   // UNICODE_TO_GBK[39826] := 16#98FC;
   // UNICODE_TO_GBK[39827] := 16#EF95;
   // UNICODE_TO_GBK[39828] := 16#98FD;
   // UNICODE_TO_GBK[39829] := 16#EF96;
   // UNICODE_TO_GBK[39830] := 16#98FE;
   // UNICODE_TO_GBK[39831] := 16#EF97;
   // UNICODE_TO_GBK[39832] := 16#98FF;
   // UNICODE_TO_GBK[39833] := 16#EF98;
   // UNICODE_TO_GBK[39834] := 16#9900;
   // UNICODE_TO_GBK[39835] := 16#EF99;
   // UNICODE_TO_GBK[39836] := 16#9901;
   // UNICODE_TO_GBK[39837] := 16#EF9A;
   // UNICODE_TO_GBK[39838] := 16#9902;
   // UNICODE_TO_GBK[39839] := 16#EF9B;
   // UNICODE_TO_GBK[39840] := 16#9903;
   // UNICODE_TO_GBK[39841] := 16#EF9C;
   // UNICODE_TO_GBK[39842] := 16#9904;
   // UNICODE_TO_GBK[39843] := 16#EF9D;
   // UNICODE_TO_GBK[39844] := 16#9905;
   // UNICODE_TO_GBK[39845] := 16#EF9E;
   // UNICODE_TO_GBK[39846] := 16#9906;
   // UNICODE_TO_GBK[39847] := 16#EF9F;
   // UNICODE_TO_GBK[39848] := 16#9907;
   // UNICODE_TO_GBK[39849] := 16#EFA0;
   // UNICODE_TO_GBK[39850] := 16#9908;
   // UNICODE_TO_GBK[39851] := 16#F040;
   // UNICODE_TO_GBK[39852] := 16#9909;
   // UNICODE_TO_GBK[39853] := 16#F041;
   // UNICODE_TO_GBK[39854] := 16#990A;
   // UNICODE_TO_GBK[39855] := 16#F042;
   // UNICODE_TO_GBK[39856] := 16#990B;
   // UNICODE_TO_GBK[39857] := 16#F043;
   // UNICODE_TO_GBK[39858] := 16#990C;
   // UNICODE_TO_GBK[39859] := 16#F044;
   // UNICODE_TO_GBK[39860] := 16#990D;
   // UNICODE_TO_GBK[39861] := 16#F7D0;
   // UNICODE_TO_GBK[39862] := 16#990E;
   // UNICODE_TO_GBK[39863] := 16#F045;
   // UNICODE_TO_GBK[39864] := 16#990F;
   // UNICODE_TO_GBK[39865] := 16#F046;
   // UNICODE_TO_GBK[39866] := 16#9910;
   // UNICODE_TO_GBK[39867] := 16#B2CD;
   // UNICODE_TO_GBK[39868] := 16#9911;
   // UNICODE_TO_GBK[39869] := 16#F047;
   // UNICODE_TO_GBK[39870] := 16#9912;
   // UNICODE_TO_GBK[39871] := 16#F048;
   // UNICODE_TO_GBK[39872] := 16#9913;
   // UNICODE_TO_GBK[39873] := 16#F049;
   // UNICODE_TO_GBK[39874] := 16#9914;
   // UNICODE_TO_GBK[39875] := 16#F04A;
   // UNICODE_TO_GBK[39876] := 16#9915;
   // UNICODE_TO_GBK[39877] := 16#F04B;
   // UNICODE_TO_GBK[39878] := 16#9916;
   // UNICODE_TO_GBK[39879] := 16#F04C;
   // UNICODE_TO_GBK[39880] := 16#9917;
   // UNICODE_TO_GBK[39881] := 16#F04D;
   // UNICODE_TO_GBK[39882] := 16#9918;
   // UNICODE_TO_GBK[39883] := 16#F04E;
   // UNICODE_TO_GBK[39884] := 16#9919;
   // UNICODE_TO_GBK[39885] := 16#F04F;
   // UNICODE_TO_GBK[39886] := 16#991A;
   // UNICODE_TO_GBK[39887] := 16#F050;
   // UNICODE_TO_GBK[39888] := 16#991B;
   // UNICODE_TO_GBK[39889] := 16#F051;
   // UNICODE_TO_GBK[39890] := 16#991C;
   // UNICODE_TO_GBK[39891] := 16#F052;
   // UNICODE_TO_GBK[39892] := 16#991D;
   // UNICODE_TO_GBK[39893] := 16#F053;
   // UNICODE_TO_GBK[39894] := 16#991E;
   // UNICODE_TO_GBK[39895] := 16#F054;
   // UNICODE_TO_GBK[39896] := 16#991F;
   // UNICODE_TO_GBK[39897] := 16#F055;
   // UNICODE_TO_GBK[39898] := 16#9920;
   // UNICODE_TO_GBK[39899] := 16#F056;
   // UNICODE_TO_GBK[39900] := 16#9921;
   // UNICODE_TO_GBK[39901] := 16#F057;
   // UNICODE_TO_GBK[39902] := 16#9922;
   // UNICODE_TO_GBK[39903] := 16#F058;
   // UNICODE_TO_GBK[39904] := 16#9923;
   // UNICODE_TO_GBK[39905] := 16#F059;
   // UNICODE_TO_GBK[39906] := 16#9924;
   // UNICODE_TO_GBK[39907] := 16#F05A;
   // UNICODE_TO_GBK[39908] := 16#9925;
   // UNICODE_TO_GBK[39909] := 16#F05B;
   // UNICODE_TO_GBK[39910] := 16#9926;
   // UNICODE_TO_GBK[39911] := 16#F05C;
   // UNICODE_TO_GBK[39912] := 16#9927;
   // UNICODE_TO_GBK[39913] := 16#F05D;
   // UNICODE_TO_GBK[39914] := 16#9928;
   // UNICODE_TO_GBK[39915] := 16#F05E;
   // UNICODE_TO_GBK[39916] := 16#9929;
   // UNICODE_TO_GBK[39917] := 16#F05F;
   // UNICODE_TO_GBK[39918] := 16#992A;
   // UNICODE_TO_GBK[39919] := 16#F060;
   // UNICODE_TO_GBK[39920] := 16#992B;
   // UNICODE_TO_GBK[39921] := 16#F061;
   // UNICODE_TO_GBK[39922] := 16#992C;
   // UNICODE_TO_GBK[39923] := 16#F062;
   // UNICODE_TO_GBK[39924] := 16#992D;
   // UNICODE_TO_GBK[39925] := 16#F063;
   // UNICODE_TO_GBK[39926] := 16#992E;
   // UNICODE_TO_GBK[39927] := 16#F7D1;
   // UNICODE_TO_GBK[39928] := 16#992F;
   // UNICODE_TO_GBK[39929] := 16#F064;
   // UNICODE_TO_GBK[39930] := 16#9930;
   // UNICODE_TO_GBK[39931] := 16#F065;
   // UNICODE_TO_GBK[39932] := 16#9931;
   // UNICODE_TO_GBK[39933] := 16#F066;
   // UNICODE_TO_GBK[39934] := 16#9932;
   // UNICODE_TO_GBK[39935] := 16#F067;
   // UNICODE_TO_GBK[39936] := 16#9933;
   // UNICODE_TO_GBK[39937] := 16#F068;
   // UNICODE_TO_GBK[39938] := 16#9934;
   // UNICODE_TO_GBK[39939] := 16#F069;
   // UNICODE_TO_GBK[39940] := 16#9935;
   // UNICODE_TO_GBK[39941] := 16#F06A;
   // UNICODE_TO_GBK[39942] := 16#9936;
   // UNICODE_TO_GBK[39943] := 16#F06B;
   // UNICODE_TO_GBK[39944] := 16#9937;
   // UNICODE_TO_GBK[39945] := 16#F06C;
   // UNICODE_TO_GBK[39946] := 16#9938;
   // UNICODE_TO_GBK[39947] := 16#F06D;
   // UNICODE_TO_GBK[39948] := 16#9939;
   // UNICODE_TO_GBK[39949] := 16#F06E;
   // UNICODE_TO_GBK[39950] := 16#993A;
   // UNICODE_TO_GBK[39951] := 16#F06F;
   // UNICODE_TO_GBK[39952] := 16#993B;
   // UNICODE_TO_GBK[39953] := 16#F070;
   // UNICODE_TO_GBK[39954] := 16#993C;
   // UNICODE_TO_GBK[39955] := 16#F071;
   // UNICODE_TO_GBK[39956] := 16#993D;
   // UNICODE_TO_GBK[39957] := 16#F072;
   // UNICODE_TO_GBK[39958] := 16#993E;
   // UNICODE_TO_GBK[39959] := 16#F073;
   // UNICODE_TO_GBK[39960] := 16#993F;
   // UNICODE_TO_GBK[39961] := 16#F074;
   // UNICODE_TO_GBK[39962] := 16#9940;
   // UNICODE_TO_GBK[39963] := 16#F075;
   // UNICODE_TO_GBK[39964] := 16#9941;
   // UNICODE_TO_GBK[39965] := 16#F076;
   // UNICODE_TO_GBK[39966] := 16#9942;
   // UNICODE_TO_GBK[39967] := 16#F077;
   // UNICODE_TO_GBK[39968] := 16#9943;
   // UNICODE_TO_GBK[39969] := 16#F078;
   // UNICODE_TO_GBK[39970] := 16#9944;
   // UNICODE_TO_GBK[39971] := 16#F079;
   // UNICODE_TO_GBK[39972] := 16#9945;
   // UNICODE_TO_GBK[39973] := 16#F07A;
   // UNICODE_TO_GBK[39974] := 16#9946;
   // UNICODE_TO_GBK[39975] := 16#F07B;
   // UNICODE_TO_GBK[39976] := 16#9947;
   // UNICODE_TO_GBK[39977] := 16#F07C;
   // UNICODE_TO_GBK[39978] := 16#9948;
   // UNICODE_TO_GBK[39979] := 16#F07D;
   // UNICODE_TO_GBK[39980] := 16#9949;
   // UNICODE_TO_GBK[39981] := 16#F07E;
   // UNICODE_TO_GBK[39982] := 16#994A;
   // UNICODE_TO_GBK[39983] := 16#F080;
   // UNICODE_TO_GBK[39984] := 16#994B;
   // UNICODE_TO_GBK[39985] := 16#F081;
   // UNICODE_TO_GBK[39986] := 16#994C;
   // UNICODE_TO_GBK[39987] := 16#F082;
   // UNICODE_TO_GBK[39988] := 16#994D;
   // UNICODE_TO_GBK[39989] := 16#F083;
   // UNICODE_TO_GBK[39990] := 16#994E;
   // UNICODE_TO_GBK[39991] := 16#F084;
   // UNICODE_TO_GBK[39992] := 16#994F;
   // UNICODE_TO_GBK[39993] := 16#F085;
   // UNICODE_TO_GBK[39994] := 16#9950;
   // UNICODE_TO_GBK[39995] := 16#F086;
   // UNICODE_TO_GBK[39996] := 16#9951;
   // UNICODE_TO_GBK[39997] := 16#F087;
   // UNICODE_TO_GBK[39998] := 16#9952;
   // UNICODE_TO_GBK[39999] := 16#F088;
   // UNICODE_TO_GBK[40000] := 16#9953;
   // UNICODE_TO_GBK[40001] := 16#F089;
   // UNICODE_TO_GBK[40002] := 16#9954;
   // UNICODE_TO_GBK[40003] := 16#F7D3;
   // UNICODE_TO_GBK[40004] := 16#9955;
   // UNICODE_TO_GBK[40005] := 16#F7D2;
   // UNICODE_TO_GBK[40006] := 16#9956;
   // UNICODE_TO_GBK[40007] := 16#F08A;
   // UNICODE_TO_GBK[40008] := 16#9957;
   // UNICODE_TO_GBK[40009] := 16#F08B;
   // UNICODE_TO_GBK[40010] := 16#9958;
   // UNICODE_TO_GBK[40011] := 16#F08C;
   // UNICODE_TO_GBK[40012] := 16#9959;
   // UNICODE_TO_GBK[40013] := 16#F08D;
   // UNICODE_TO_GBK[40014] := 16#995A;
   // UNICODE_TO_GBK[40015] := 16#F08E;
   // UNICODE_TO_GBK[40016] := 16#995B;
   // UNICODE_TO_GBK[40017] := 16#F08F;
   // UNICODE_TO_GBK[40018] := 16#995C;
   // UNICODE_TO_GBK[40019] := 16#F090;
   // UNICODE_TO_GBK[40020] := 16#995D;
   // UNICODE_TO_GBK[40021] := 16#F091;
   // UNICODE_TO_GBK[40022] := 16#995E;
   // UNICODE_TO_GBK[40023] := 16#F092;
   // UNICODE_TO_GBK[40024] := 16#995F;
   // UNICODE_TO_GBK[40025] := 16#F093;
   // UNICODE_TO_GBK[40026] := 16#9960;
   // UNICODE_TO_GBK[40027] := 16#F094;
   // UNICODE_TO_GBK[40028] := 16#9961;
   // UNICODE_TO_GBK[40029] := 16#F095;
   // UNICODE_TO_GBK[40030] := 16#9962;
   // UNICODE_TO_GBK[40031] := 16#F096;
   // UNICODE_TO_GBK[40032] := 16#9963;
   // UNICODE_TO_GBK[40033] := 16#E2BB;
   // UNICODE_TO_GBK[40034] := 16#9964;
   // UNICODE_TO_GBK[40035] := 16#F097;
   // UNICODE_TO_GBK[40036] := 16#9965;
   // UNICODE_TO_GBK[40037] := 16#BCA2;
   // UNICODE_TO_GBK[40038] := 16#9966;
   // UNICODE_TO_GBK[40039] := 16#F098;
   // UNICODE_TO_GBK[40040] := 16#9967;
   // UNICODE_TO_GBK[40041] := 16#E2BC;
   // UNICODE_TO_GBK[40042] := 16#9968;
   // UNICODE_TO_GBK[40043] := 16#E2BD;
   // UNICODE_TO_GBK[40044] := 16#9969;
   // UNICODE_TO_GBK[40045] := 16#E2BE;
   // UNICODE_TO_GBK[40046] := 16#996A;
   // UNICODE_TO_GBK[40047] := 16#E2BF;
   // UNICODE_TO_GBK[40048] := 16#996B;
   // UNICODE_TO_GBK[40049] := 16#E2C0;
   // UNICODE_TO_GBK[40050] := 16#996C;
   // UNICODE_TO_GBK[40051] := 16#E2C1;
   // UNICODE_TO_GBK[40052] := 16#996D;
   // UNICODE_TO_GBK[40053] := 16#B7B9;
   // UNICODE_TO_GBK[40054] := 16#996E;
   // UNICODE_TO_GBK[40055] := 16#D2FB;
   // UNICODE_TO_GBK[40056] := 16#996F;
   // UNICODE_TO_GBK[40057] := 16#BDA4;
   // UNICODE_TO_GBK[40058] := 16#9970;
   // UNICODE_TO_GBK[40059] := 16#CACE;
   // UNICODE_TO_GBK[40060] := 16#9971;
   // UNICODE_TO_GBK[40061] := 16#B1A5;
   // UNICODE_TO_GBK[40062] := 16#9972;
   // UNICODE_TO_GBK[40063] := 16#CBC7;
   // UNICODE_TO_GBK[40064] := 16#9973;
   // UNICODE_TO_GBK[40065] := 16#F099;
   // UNICODE_TO_GBK[40066] := 16#9974;
   // UNICODE_TO_GBK[40067] := 16#E2C2;
   // UNICODE_TO_GBK[40068] := 16#9975;
   // UNICODE_TO_GBK[40069] := 16#B6FC;
   // UNICODE_TO_GBK[40070] := 16#9976;
   // UNICODE_TO_GBK[40071] := 16#C8C4;
   // UNICODE_TO_GBK[40072] := 16#9977;
   // UNICODE_TO_GBK[40073] := 16#E2C3;
   // UNICODE_TO_GBK[40074] := 16#9978;
   // UNICODE_TO_GBK[40075] := 16#F09A;
   // UNICODE_TO_GBK[40076] := 16#9979;
   // UNICODE_TO_GBK[40077] := 16#F09B;
   // UNICODE_TO_GBK[40078] := 16#997A;
   // UNICODE_TO_GBK[40079] := 16#BDC8;
   // UNICODE_TO_GBK[40080] := 16#997B;
   // UNICODE_TO_GBK[40081] := 16#F09C;
   // UNICODE_TO_GBK[40082] := 16#997C;
   // UNICODE_TO_GBK[40083] := 16#B1FD;
   // UNICODE_TO_GBK[40084] := 16#997D;
   // UNICODE_TO_GBK[40085] := 16#E2C4;
   // UNICODE_TO_GBK[40086] := 16#997E;
   // UNICODE_TO_GBK[40087] := 16#F09D;
   // UNICODE_TO_GBK[40088] := 16#997F;
   // UNICODE_TO_GBK[40089] := 16#B6F6;
   // UNICODE_TO_GBK[40090] := 16#9980;
   // UNICODE_TO_GBK[40091] := 16#E2C5;
   // UNICODE_TO_GBK[40092] := 16#9981;
   // UNICODE_TO_GBK[40093] := 16#C4D9;
   // UNICODE_TO_GBK[40094] := 16#9982;
   // UNICODE_TO_GBK[40095] := 16#F09E;
   // UNICODE_TO_GBK[40096] := 16#9983;
   // UNICODE_TO_GBK[40097] := 16#F09F;
   // UNICODE_TO_GBK[40098] := 16#9984;
   // UNICODE_TO_GBK[40099] := 16#E2C6;
   // UNICODE_TO_GBK[40100] := 16#9985;
   // UNICODE_TO_GBK[40101] := 16#CFDA;
   // UNICODE_TO_GBK[40102] := 16#9986;
   // UNICODE_TO_GBK[40103] := 16#B9DD;
   // UNICODE_TO_GBK[40104] := 16#9987;
   // UNICODE_TO_GBK[40105] := 16#E2C7;
   // UNICODE_TO_GBK[40106] := 16#9988;
   // UNICODE_TO_GBK[40107] := 16#C0A1;
   // UNICODE_TO_GBK[40108] := 16#9989;
   // UNICODE_TO_GBK[40109] := 16#F0A0;
   // UNICODE_TO_GBK[40110] := 16#998A;
   // UNICODE_TO_GBK[40111] := 16#E2C8;
   // UNICODE_TO_GBK[40112] := 16#998B;
   // UNICODE_TO_GBK[40113] := 16#B2F6;
   // UNICODE_TO_GBK[40114] := 16#998C;
   // UNICODE_TO_GBK[40115] := 16#F140;
   // UNICODE_TO_GBK[40116] := 16#998D;
   // UNICODE_TO_GBK[40117] := 16#E2C9;
   // UNICODE_TO_GBK[40118] := 16#998E;
   // UNICODE_TO_GBK[40119] := 16#F141;
   // UNICODE_TO_GBK[40120] := 16#998F;
   // UNICODE_TO_GBK[40121] := 16#C1F3;
   // UNICODE_TO_GBK[40122] := 16#9990;
   // UNICODE_TO_GBK[40123] := 16#E2CA;
   // UNICODE_TO_GBK[40124] := 16#9991;
   // UNICODE_TO_GBK[40125] := 16#E2CB;
   // UNICODE_TO_GBK[40126] := 16#9992;
   // UNICODE_TO_GBK[40127] := 16#C2F8;
   // UNICODE_TO_GBK[40128] := 16#9993;
   // UNICODE_TO_GBK[40129] := 16#E2CC;
   // UNICODE_TO_GBK[40130] := 16#9994;
   // UNICODE_TO_GBK[40131] := 16#E2CD;
   // UNICODE_TO_GBK[40132] := 16#9995;
   // UNICODE_TO_GBK[40133] := 16#E2CE;
   // UNICODE_TO_GBK[40134] := 16#9996;
   // UNICODE_TO_GBK[40135] := 16#CAD7;
   // UNICODE_TO_GBK[40136] := 16#9997;
   // UNICODE_TO_GBK[40137] := 16#D8B8;
   // UNICODE_TO_GBK[40138] := 16#9998;
   // UNICODE_TO_GBK[40139] := 16#D9E5;
   // UNICODE_TO_GBK[40140] := 16#9999;
   // UNICODE_TO_GBK[40141] := 16#CFE3;
   // UNICODE_TO_GBK[40142] := 16#999A;
   // UNICODE_TO_GBK[40143] := 16#F142;
   // UNICODE_TO_GBK[40144] := 16#999B;
   // UNICODE_TO_GBK[40145] := 16#F143;
   // UNICODE_TO_GBK[40146] := 16#999C;
   // UNICODE_TO_GBK[40147] := 16#F144;
   // UNICODE_TO_GBK[40148] := 16#999D;
   // UNICODE_TO_GBK[40149] := 16#F145;
   // UNICODE_TO_GBK[40150] := 16#999E;
   // UNICODE_TO_GBK[40151] := 16#F146;
   // UNICODE_TO_GBK[40152] := 16#999F;
   // UNICODE_TO_GBK[40153] := 16#F147;
   // UNICODE_TO_GBK[40154] := 16#99A0;
   // UNICODE_TO_GBK[40155] := 16#F148;
   // UNICODE_TO_GBK[40156] := 16#99A1;
   // UNICODE_TO_GBK[40157] := 16#F149;
   // UNICODE_TO_GBK[40158] := 16#99A2;
   // UNICODE_TO_GBK[40159] := 16#F14A;
   // UNICODE_TO_GBK[40160] := 16#99A3;
   // UNICODE_TO_GBK[40161] := 16#F14B;
   // UNICODE_TO_GBK[40162] := 16#99A4;
   // UNICODE_TO_GBK[40163] := 16#F14C;
   // UNICODE_TO_GBK[40164] := 16#99A5;
   // UNICODE_TO_GBK[40165] := 16#F0A5;
   // UNICODE_TO_GBK[40166] := 16#99A6;
   // UNICODE_TO_GBK[40167] := 16#F14D;
   // UNICODE_TO_GBK[40168] := 16#99A7;
   // UNICODE_TO_GBK[40169] := 16#F14E;
   // UNICODE_TO_GBK[40170] := 16#99A8;
   // UNICODE_TO_GBK[40171] := 16#DCB0;
   // UNICODE_TO_GBK[40172] := 16#99A9;
   // UNICODE_TO_GBK[40173] := 16#F14F;
   // UNICODE_TO_GBK[40174] := 16#99AA;
   // UNICODE_TO_GBK[40175] := 16#F150;
   // UNICODE_TO_GBK[40176] := 16#99AB;
   // UNICODE_TO_GBK[40177] := 16#F151;
   // UNICODE_TO_GBK[40178] := 16#99AC;
   // UNICODE_TO_GBK[40179] := 16#F152;
   // UNICODE_TO_GBK[40180] := 16#99AD;
   // UNICODE_TO_GBK[40181] := 16#F153;
   // UNICODE_TO_GBK[40182] := 16#99AE;
   // UNICODE_TO_GBK[40183] := 16#F154;
   // UNICODE_TO_GBK[40184] := 16#99AF;
   // UNICODE_TO_GBK[40185] := 16#F155;
   // UNICODE_TO_GBK[40186] := 16#99B0;
   // UNICODE_TO_GBK[40187] := 16#F156;
   // UNICODE_TO_GBK[40188] := 16#99B1;
   // UNICODE_TO_GBK[40189] := 16#F157;
   // UNICODE_TO_GBK[40190] := 16#99B2;
   // UNICODE_TO_GBK[40191] := 16#F158;
   // UNICODE_TO_GBK[40192] := 16#99B3;
   // UNICODE_TO_GBK[40193] := 16#F159;
   // UNICODE_TO_GBK[40194] := 16#99B4;
   // UNICODE_TO_GBK[40195] := 16#F15A;
   // UNICODE_TO_GBK[40196] := 16#99B5;
   // UNICODE_TO_GBK[40197] := 16#F15B;
   // UNICODE_TO_GBK[40198] := 16#99B6;
   // UNICODE_TO_GBK[40199] := 16#F15C;
   // UNICODE_TO_GBK[40200] := 16#99B7;
   // UNICODE_TO_GBK[40201] := 16#F15D;
   // UNICODE_TO_GBK[40202] := 16#99B8;
   // UNICODE_TO_GBK[40203] := 16#F15E;
   // UNICODE_TO_GBK[40204] := 16#99B9;
   // UNICODE_TO_GBK[40205] := 16#F15F;
   // UNICODE_TO_GBK[40206] := 16#99BA;
   // UNICODE_TO_GBK[40207] := 16#F160;
   // UNICODE_TO_GBK[40208] := 16#99BB;
   // UNICODE_TO_GBK[40209] := 16#F161;
   // UNICODE_TO_GBK[40210] := 16#99BC;
   // UNICODE_TO_GBK[40211] := 16#F162;
   // UNICODE_TO_GBK[40212] := 16#99BD;
   // UNICODE_TO_GBK[40213] := 16#F163;
   // UNICODE_TO_GBK[40214] := 16#99BE;
   // UNICODE_TO_GBK[40215] := 16#F164;
   // UNICODE_TO_GBK[40216] := 16#99BF;
   // UNICODE_TO_GBK[40217] := 16#F165;
   // UNICODE_TO_GBK[40218] := 16#99C0;
   // UNICODE_TO_GBK[40219] := 16#F166;
   // UNICODE_TO_GBK[40220] := 16#99C1;
   // UNICODE_TO_GBK[40221] := 16#F167;
   // UNICODE_TO_GBK[40222] := 16#99C2;
   // UNICODE_TO_GBK[40223] := 16#F168;
   // UNICODE_TO_GBK[40224] := 16#99C3;
   // UNICODE_TO_GBK[40225] := 16#F169;
   // UNICODE_TO_GBK[40226] := 16#99C4;
   // UNICODE_TO_GBK[40227] := 16#F16A;
   // UNICODE_TO_GBK[40228] := 16#99C5;
   // UNICODE_TO_GBK[40229] := 16#F16B;
   // UNICODE_TO_GBK[40230] := 16#99C6;
   // UNICODE_TO_GBK[40231] := 16#F16C;
   // UNICODE_TO_GBK[40232] := 16#99C7;
   // UNICODE_TO_GBK[40233] := 16#F16D;
   // UNICODE_TO_GBK[40234] := 16#99C8;
   // UNICODE_TO_GBK[40235] := 16#F16E;
   // UNICODE_TO_GBK[40236] := 16#99C9;
   // UNICODE_TO_GBK[40237] := 16#F16F;
   // UNICODE_TO_GBK[40238] := 16#99CA;
   // UNICODE_TO_GBK[40239] := 16#F170;
   // UNICODE_TO_GBK[40240] := 16#99CB;
   // UNICODE_TO_GBK[40241] := 16#F171;
   // UNICODE_TO_GBK[40242] := 16#99CC;
   // UNICODE_TO_GBK[40243] := 16#F172;
   // UNICODE_TO_GBK[40244] := 16#99CD;
   // UNICODE_TO_GBK[40245] := 16#F173;
   // UNICODE_TO_GBK[40246] := 16#99CE;
   // UNICODE_TO_GBK[40247] := 16#F174;
   // UNICODE_TO_GBK[40248] := 16#99CF;
   // UNICODE_TO_GBK[40249] := 16#F175;
   // UNICODE_TO_GBK[40250] := 16#99D0;
   // UNICODE_TO_GBK[40251] := 16#F176;
   // UNICODE_TO_GBK[40252] := 16#99D1;
   // UNICODE_TO_GBK[40253] := 16#F177;
   // UNICODE_TO_GBK[40254] := 16#99D2;
   // UNICODE_TO_GBK[40255] := 16#F178;
   // UNICODE_TO_GBK[40256] := 16#99D3;
   // UNICODE_TO_GBK[40257] := 16#F179;
   // UNICODE_TO_GBK[40258] := 16#99D4;
   // UNICODE_TO_GBK[40259] := 16#F17A;
   // UNICODE_TO_GBK[40260] := 16#99D5;
   // UNICODE_TO_GBK[40261] := 16#F17B;
   // UNICODE_TO_GBK[40262] := 16#99D6;
   // UNICODE_TO_GBK[40263] := 16#F17C;
   // UNICODE_TO_GBK[40264] := 16#99D7;
   // UNICODE_TO_GBK[40265] := 16#F17D;
   // UNICODE_TO_GBK[40266] := 16#99D8;
   // UNICODE_TO_GBK[40267] := 16#F17E;
   // UNICODE_TO_GBK[40268] := 16#99D9;
   // UNICODE_TO_GBK[40269] := 16#F180;
   // UNICODE_TO_GBK[40270] := 16#99DA;
   // UNICODE_TO_GBK[40271] := 16#F181;
   // UNICODE_TO_GBK[40272] := 16#99DB;
   // UNICODE_TO_GBK[40273] := 16#F182;
   // UNICODE_TO_GBK[40274] := 16#99DC;
   // UNICODE_TO_GBK[40275] := 16#F183;
   // UNICODE_TO_GBK[40276] := 16#99DD;
   // UNICODE_TO_GBK[40277] := 16#F184;
   // UNICODE_TO_GBK[40278] := 16#99DE;
   // UNICODE_TO_GBK[40279] := 16#F185;
   // UNICODE_TO_GBK[40280] := 16#99DF;
   // UNICODE_TO_GBK[40281] := 16#F186;
   // UNICODE_TO_GBK[40282] := 16#99E0;
   // UNICODE_TO_GBK[40283] := 16#F187;
   // UNICODE_TO_GBK[40284] := 16#99E1;
   // UNICODE_TO_GBK[40285] := 16#F188;
   // UNICODE_TO_GBK[40286] := 16#99E2;
   // UNICODE_TO_GBK[40287] := 16#F189;
   // UNICODE_TO_GBK[40288] := 16#99E3;
   // UNICODE_TO_GBK[40289] := 16#F18A;
   // UNICODE_TO_GBK[40290] := 16#99E4;
   // UNICODE_TO_GBK[40291] := 16#F18B;
   // UNICODE_TO_GBK[40292] := 16#99E5;
   // UNICODE_TO_GBK[40293] := 16#F18C;
   // UNICODE_TO_GBK[40294] := 16#99E6;
   // UNICODE_TO_GBK[40295] := 16#F18D;
   // UNICODE_TO_GBK[40296] := 16#99E7;
   // UNICODE_TO_GBK[40297] := 16#F18E;
   // UNICODE_TO_GBK[40298] := 16#99E8;
   // UNICODE_TO_GBK[40299] := 16#F18F;
   // UNICODE_TO_GBK[40300] := 16#99E9;
   // UNICODE_TO_GBK[40301] := 16#F190;
   // UNICODE_TO_GBK[40302] := 16#99EA;
   // UNICODE_TO_GBK[40303] := 16#F191;
   // UNICODE_TO_GBK[40304] := 16#99EB;
   // UNICODE_TO_GBK[40305] := 16#F192;
   // UNICODE_TO_GBK[40306] := 16#99EC;
   // UNICODE_TO_GBK[40307] := 16#F193;
   // UNICODE_TO_GBK[40308] := 16#99ED;
   // UNICODE_TO_GBK[40309] := 16#F194;
   // UNICODE_TO_GBK[40310] := 16#99EE;
   // UNICODE_TO_GBK[40311] := 16#F195;
   // UNICODE_TO_GBK[40312] := 16#99EF;
   // UNICODE_TO_GBK[40313] := 16#F196;
   // UNICODE_TO_GBK[40314] := 16#99F0;
   // UNICODE_TO_GBK[40315] := 16#F197;
   // UNICODE_TO_GBK[40316] := 16#99F1;
   // UNICODE_TO_GBK[40317] := 16#F198;
   // UNICODE_TO_GBK[40318] := 16#99F2;
   // UNICODE_TO_GBK[40319] := 16#F199;
   // UNICODE_TO_GBK[40320] := 16#99F3;
   // UNICODE_TO_GBK[40321] := 16#F19A;
   // UNICODE_TO_GBK[40322] := 16#99F4;
   // UNICODE_TO_GBK[40323] := 16#F19B;
   // UNICODE_TO_GBK[40324] := 16#99F5;
   // UNICODE_TO_GBK[40325] := 16#F19C;
   // UNICODE_TO_GBK[40326] := 16#99F6;
   // UNICODE_TO_GBK[40327] := 16#F19D;
   // UNICODE_TO_GBK[40328] := 16#99F7;
   // UNICODE_TO_GBK[40329] := 16#F19E;
   // UNICODE_TO_GBK[40330] := 16#99F8;
   // UNICODE_TO_GBK[40331] := 16#F19F;
   // UNICODE_TO_GBK[40332] := 16#99F9;
   // UNICODE_TO_GBK[40333] := 16#F1A0;
   // UNICODE_TO_GBK[40334] := 16#99FA;
   // UNICODE_TO_GBK[40335] := 16#F240;
   // UNICODE_TO_GBK[40336] := 16#99FB;
   // UNICODE_TO_GBK[40337] := 16#F241;
   // UNICODE_TO_GBK[40338] := 16#99FC;
   // UNICODE_TO_GBK[40339] := 16#F242;
   // UNICODE_TO_GBK[40340] := 16#99FD;
   // UNICODE_TO_GBK[40341] := 16#F243;
   // UNICODE_TO_GBK[40342] := 16#99FE;
   // UNICODE_TO_GBK[40343] := 16#F244;
   // UNICODE_TO_GBK[40344] := 16#99FF;
   // UNICODE_TO_GBK[40345] := 16#F245;
   // UNICODE_TO_GBK[40346] := 16#9A00;
   // UNICODE_TO_GBK[40347] := 16#F246;
   // UNICODE_TO_GBK[40348] := 16#9A01;
   // UNICODE_TO_GBK[40349] := 16#F247;
   // UNICODE_TO_GBK[40350] := 16#9A02;
   // UNICODE_TO_GBK[40351] := 16#F248;
   // UNICODE_TO_GBK[40352] := 16#9A03;
   // UNICODE_TO_GBK[40353] := 16#F249;
   // UNICODE_TO_GBK[40354] := 16#9A04;
   // UNICODE_TO_GBK[40355] := 16#F24A;
   // UNICODE_TO_GBK[40356] := 16#9A05;
   // UNICODE_TO_GBK[40357] := 16#F24B;
   // UNICODE_TO_GBK[40358] := 16#9A06;
   // UNICODE_TO_GBK[40359] := 16#F24C;
   // UNICODE_TO_GBK[40360] := 16#9A07;
   // UNICODE_TO_GBK[40361] := 16#F24D;
   // UNICODE_TO_GBK[40362] := 16#9A08;
   // UNICODE_TO_GBK[40363] := 16#F24E;
   // UNICODE_TO_GBK[40364] := 16#9A09;
   // UNICODE_TO_GBK[40365] := 16#F24F;
   // UNICODE_TO_GBK[40366] := 16#9A0A;
   // UNICODE_TO_GBK[40367] := 16#F250;
   // UNICODE_TO_GBK[40368] := 16#9A0B;
   // UNICODE_TO_GBK[40369] := 16#F251;
   // UNICODE_TO_GBK[40370] := 16#9A0C;
   // UNICODE_TO_GBK[40371] := 16#F252;
   // UNICODE_TO_GBK[40372] := 16#9A0D;
   // UNICODE_TO_GBK[40373] := 16#F253;
   // UNICODE_TO_GBK[40374] := 16#9A0E;
   // UNICODE_TO_GBK[40375] := 16#F254;
   // UNICODE_TO_GBK[40376] := 16#9A0F;
   // UNICODE_TO_GBK[40377] := 16#F255;
   // UNICODE_TO_GBK[40378] := 16#9A10;
   // UNICODE_TO_GBK[40379] := 16#F256;
   // UNICODE_TO_GBK[40380] := 16#9A11;
   // UNICODE_TO_GBK[40381] := 16#F257;
   // UNICODE_TO_GBK[40382] := 16#9A12;
   // UNICODE_TO_GBK[40383] := 16#F258;
   // UNICODE_TO_GBK[40384] := 16#9A13;
   // UNICODE_TO_GBK[40385] := 16#F259;
   // UNICODE_TO_GBK[40386] := 16#9A14;
   // UNICODE_TO_GBK[40387] := 16#F25A;
   // UNICODE_TO_GBK[40388] := 16#9A15;
   // UNICODE_TO_GBK[40389] := 16#F25B;
   // UNICODE_TO_GBK[40390] := 16#9A16;
   // UNICODE_TO_GBK[40391] := 16#F25C;
   // UNICODE_TO_GBK[40392] := 16#9A17;
   // UNICODE_TO_GBK[40393] := 16#F25D;
   // UNICODE_TO_GBK[40394] := 16#9A18;
   // UNICODE_TO_GBK[40395] := 16#F25E;
   // UNICODE_TO_GBK[40396] := 16#9A19;
   // UNICODE_TO_GBK[40397] := 16#F25F;
   // UNICODE_TO_GBK[40398] := 16#9A1A;
   // UNICODE_TO_GBK[40399] := 16#F260;
   // UNICODE_TO_GBK[40400] := 16#9A1B;
   // UNICODE_TO_GBK[40401] := 16#F261;
   // UNICODE_TO_GBK[40402] := 16#9A1C;
   // UNICODE_TO_GBK[40403] := 16#F262;
   // UNICODE_TO_GBK[40404] := 16#9A1D;
   // UNICODE_TO_GBK[40405] := 16#F263;
   // UNICODE_TO_GBK[40406] := 16#9A1E;
   // UNICODE_TO_GBK[40407] := 16#F264;
   // UNICODE_TO_GBK[40408] := 16#9A1F;
   // UNICODE_TO_GBK[40409] := 16#F265;
   // UNICODE_TO_GBK[40410] := 16#9A20;
   // UNICODE_TO_GBK[40411] := 16#F266;
   // UNICODE_TO_GBK[40412] := 16#9A21;
   // UNICODE_TO_GBK[40413] := 16#F267;
   // UNICODE_TO_GBK[40414] := 16#9A22;
   // UNICODE_TO_GBK[40415] := 16#F268;
   // UNICODE_TO_GBK[40416] := 16#9A23;
   // UNICODE_TO_GBK[40417] := 16#F269;
   // UNICODE_TO_GBK[40418] := 16#9A24;
   // UNICODE_TO_GBK[40419] := 16#F26A;
   // UNICODE_TO_GBK[40420] := 16#9A25;
   // UNICODE_TO_GBK[40421] := 16#F26B;
   // UNICODE_TO_GBK[40422] := 16#9A26;
   // UNICODE_TO_GBK[40423] := 16#F26C;
   // UNICODE_TO_GBK[40424] := 16#9A27;
   // UNICODE_TO_GBK[40425] := 16#F26D;
   // UNICODE_TO_GBK[40426] := 16#9A28;
   // UNICODE_TO_GBK[40427] := 16#F26E;
   // UNICODE_TO_GBK[40428] := 16#9A29;
   // UNICODE_TO_GBK[40429] := 16#F26F;
   // UNICODE_TO_GBK[40430] := 16#9A2A;
   // UNICODE_TO_GBK[40431] := 16#F270;
   // UNICODE_TO_GBK[40432] := 16#9A2B;
   // UNICODE_TO_GBK[40433] := 16#F271;
   // UNICODE_TO_GBK[40434] := 16#9A2C;
   // UNICODE_TO_GBK[40435] := 16#F272;
   // UNICODE_TO_GBK[40436] := 16#9A2D;
   // UNICODE_TO_GBK[40437] := 16#F273;
   // UNICODE_TO_GBK[40438] := 16#9A2E;
   // UNICODE_TO_GBK[40439] := 16#F274;
   // UNICODE_TO_GBK[40440] := 16#9A2F;
   // UNICODE_TO_GBK[40441] := 16#F275;
   // UNICODE_TO_GBK[40442] := 16#9A30;
   // UNICODE_TO_GBK[40443] := 16#F276;
   // UNICODE_TO_GBK[40444] := 16#9A31;
   // UNICODE_TO_GBK[40445] := 16#F277;
   // UNICODE_TO_GBK[40446] := 16#9A32;
   // UNICODE_TO_GBK[40447] := 16#F278;
   // UNICODE_TO_GBK[40448] := 16#9A33;
   // UNICODE_TO_GBK[40449] := 16#F279;
   // UNICODE_TO_GBK[40450] := 16#9A34;
   // UNICODE_TO_GBK[40451] := 16#F27A;
   // UNICODE_TO_GBK[40452] := 16#9A35;
   // UNICODE_TO_GBK[40453] := 16#F27B;
   // UNICODE_TO_GBK[40454] := 16#9A36;
   // UNICODE_TO_GBK[40455] := 16#F27C;
   // UNICODE_TO_GBK[40456] := 16#9A37;
   // UNICODE_TO_GBK[40457] := 16#F27D;
   // UNICODE_TO_GBK[40458] := 16#9A38;
   // UNICODE_TO_GBK[40459] := 16#F27E;
   // UNICODE_TO_GBK[40460] := 16#9A39;
   // UNICODE_TO_GBK[40461] := 16#F280;
   // UNICODE_TO_GBK[40462] := 16#9A3A;
   // UNICODE_TO_GBK[40463] := 16#F281;
   // UNICODE_TO_GBK[40464] := 16#9A3B;
   // UNICODE_TO_GBK[40465] := 16#F282;
   // UNICODE_TO_GBK[40466] := 16#9A3C;
   // UNICODE_TO_GBK[40467] := 16#F283;
   // UNICODE_TO_GBK[40468] := 16#9A3D;
   // UNICODE_TO_GBK[40469] := 16#F284;
   // UNICODE_TO_GBK[40470] := 16#9A3E;
   // UNICODE_TO_GBK[40471] := 16#F285;
   // UNICODE_TO_GBK[40472] := 16#9A3F;
   // UNICODE_TO_GBK[40473] := 16#F286;
   // UNICODE_TO_GBK[40474] := 16#9A40;
   // UNICODE_TO_GBK[40475] := 16#F287;
   // UNICODE_TO_GBK[40476] := 16#9A41;
   // UNICODE_TO_GBK[40477] := 16#F288;
   // UNICODE_TO_GBK[40478] := 16#9A42;
   // UNICODE_TO_GBK[40479] := 16#F289;
   // UNICODE_TO_GBK[40480] := 16#9A43;
   // UNICODE_TO_GBK[40481] := 16#F28A;
   // UNICODE_TO_GBK[40482] := 16#9A44;
   // UNICODE_TO_GBK[40483] := 16#F28B;
   // UNICODE_TO_GBK[40484] := 16#9A45;
   // UNICODE_TO_GBK[40485] := 16#F28C;
   // UNICODE_TO_GBK[40486] := 16#9A46;
   // UNICODE_TO_GBK[40487] := 16#F28D;
   // UNICODE_TO_GBK[40488] := 16#9A47;
   // UNICODE_TO_GBK[40489] := 16#F28E;
   // UNICODE_TO_GBK[40490] := 16#9A48;
   // UNICODE_TO_GBK[40491] := 16#F28F;
   // UNICODE_TO_GBK[40492] := 16#9A49;
   // UNICODE_TO_GBK[40493] := 16#F290;
   // UNICODE_TO_GBK[40494] := 16#9A4A;
   // UNICODE_TO_GBK[40495] := 16#F291;
   // UNICODE_TO_GBK[40496] := 16#9A4B;
   // UNICODE_TO_GBK[40497] := 16#F292;
   // UNICODE_TO_GBK[40498] := 16#9A4C;
   // UNICODE_TO_GBK[40499] := 16#F293;
   // UNICODE_TO_GBK[40500] := 16#9A4D;
   // UNICODE_TO_GBK[40501] := 16#F294;
   // UNICODE_TO_GBK[40502] := 16#9A4E;
   // UNICODE_TO_GBK[40503] := 16#F295;
   // UNICODE_TO_GBK[40504] := 16#9A4F;
   // UNICODE_TO_GBK[40505] := 16#F296;
   // UNICODE_TO_GBK[40506] := 16#9A50;
   // UNICODE_TO_GBK[40507] := 16#F297;
   // UNICODE_TO_GBK[40508] := 16#9A51;
   // UNICODE_TO_GBK[40509] := 16#F298;
   // UNICODE_TO_GBK[40510] := 16#9A52;
   // UNICODE_TO_GBK[40511] := 16#F299;
   // UNICODE_TO_GBK[40512] := 16#9A53;
   // UNICODE_TO_GBK[40513] := 16#F29A;
   // UNICODE_TO_GBK[40514] := 16#9A54;
   // UNICODE_TO_GBK[40515] := 16#F29B;
   // UNICODE_TO_GBK[40516] := 16#9A55;
   // UNICODE_TO_GBK[40517] := 16#F29C;
   // UNICODE_TO_GBK[40518] := 16#9A56;
   // UNICODE_TO_GBK[40519] := 16#F29D;
   // UNICODE_TO_GBK[40520] := 16#9A57;
   // UNICODE_TO_GBK[40521] := 16#F29E;
   // UNICODE_TO_GBK[40522] := 16#9A58;
   // UNICODE_TO_GBK[40523] := 16#F29F;
   // UNICODE_TO_GBK[40524] := 16#9A59;
   // UNICODE_TO_GBK[40525] := 16#F2A0;
   // UNICODE_TO_GBK[40526] := 16#9A5A;
   // UNICODE_TO_GBK[40527] := 16#F340;
   // UNICODE_TO_GBK[40528] := 16#9A5B;
   // UNICODE_TO_GBK[40529] := 16#F341;
   // UNICODE_TO_GBK[40530] := 16#9A5C;
   // UNICODE_TO_GBK[40531] := 16#F342;
   // UNICODE_TO_GBK[40532] := 16#9A5D;
   // UNICODE_TO_GBK[40533] := 16#F343;
   // UNICODE_TO_GBK[40534] := 16#9A5E;
   // UNICODE_TO_GBK[40535] := 16#F344;
   // UNICODE_TO_GBK[40536] := 16#9A5F;
   // UNICODE_TO_GBK[40537] := 16#F345;
   // UNICODE_TO_GBK[40538] := 16#9A60;
   // UNICODE_TO_GBK[40539] := 16#F346;
   // UNICODE_TO_GBK[40540] := 16#9A61;
   // UNICODE_TO_GBK[40541] := 16#F347;
   // UNICODE_TO_GBK[40542] := 16#9A62;
   // UNICODE_TO_GBK[40543] := 16#F348;
   // UNICODE_TO_GBK[40544] := 16#9A63;
   // UNICODE_TO_GBK[40545] := 16#F349;
   // UNICODE_TO_GBK[40546] := 16#9A64;
   // UNICODE_TO_GBK[40547] := 16#F34A;
   // UNICODE_TO_GBK[40548] := 16#9A65;
   // UNICODE_TO_GBK[40549] := 16#F34B;
   // UNICODE_TO_GBK[40550] := 16#9A66;
   // UNICODE_TO_GBK[40551] := 16#F34C;
   // UNICODE_TO_GBK[40552] := 16#9A67;
   // UNICODE_TO_GBK[40553] := 16#F34D;
   // UNICODE_TO_GBK[40554] := 16#9A68;
   // UNICODE_TO_GBK[40555] := 16#F34E;
   // UNICODE_TO_GBK[40556] := 16#9A69;
   // UNICODE_TO_GBK[40557] := 16#F34F;
   // UNICODE_TO_GBK[40558] := 16#9A6A;
   // UNICODE_TO_GBK[40559] := 16#F350;
   // UNICODE_TO_GBK[40560] := 16#9A6B;
   // UNICODE_TO_GBK[40561] := 16#F351;
   // UNICODE_TO_GBK[40562] := 16#9A6C;
   // UNICODE_TO_GBK[40563] := 16#C2ED;
   // UNICODE_TO_GBK[40564] := 16#9A6D;
   // UNICODE_TO_GBK[40565] := 16#D4A6;
   // UNICODE_TO_GBK[40566] := 16#9A6E;
   // UNICODE_TO_GBK[40567] := 16#CDD4;
   // UNICODE_TO_GBK[40568] := 16#9A6F;
   // UNICODE_TO_GBK[40569] := 16#D1B1;
   // UNICODE_TO_GBK[40570] := 16#9A70;
   // UNICODE_TO_GBK[40571] := 16#B3DB;
   // UNICODE_TO_GBK[40572] := 16#9A71;
   // UNICODE_TO_GBK[40573] := 16#C7FD;
   // UNICODE_TO_GBK[40574] := 16#9A72;
   // UNICODE_TO_GBK[40575] := 16#F352;
   // UNICODE_TO_GBK[40576] := 16#9A73;
   // UNICODE_TO_GBK[40577] := 16#B2B5;
   // UNICODE_TO_GBK[40578] := 16#9A74;
   // UNICODE_TO_GBK[40579] := 16#C2BF;
   // UNICODE_TO_GBK[40580] := 16#9A75;
   // UNICODE_TO_GBK[40581] := 16#E6E0;
   // UNICODE_TO_GBK[40582] := 16#9A76;
   // UNICODE_TO_GBK[40583] := 16#CABB;
   // UNICODE_TO_GBK[40584] := 16#9A77;
   // UNICODE_TO_GBK[40585] := 16#E6E1;
   // UNICODE_TO_GBK[40586] := 16#9A78;
   // UNICODE_TO_GBK[40587] := 16#E6E2;
   // UNICODE_TO_GBK[40588] := 16#9A79;
   // UNICODE_TO_GBK[40589] := 16#BED4;
   // UNICODE_TO_GBK[40590] := 16#9A7A;
   // UNICODE_TO_GBK[40591] := 16#E6E3;
   // UNICODE_TO_GBK[40592] := 16#9A7B;
   // UNICODE_TO_GBK[40593] := 16#D7A4;
   // UNICODE_TO_GBK[40594] := 16#9A7C;
   // UNICODE_TO_GBK[40595] := 16#CDD5;
   // UNICODE_TO_GBK[40596] := 16#9A7D;
   // UNICODE_TO_GBK[40597] := 16#E6E5;
   // UNICODE_TO_GBK[40598] := 16#9A7E;
   // UNICODE_TO_GBK[40599] := 16#BCDD;
   // UNICODE_TO_GBK[40600] := 16#9A7F;
   // UNICODE_TO_GBK[40601] := 16#E6E4;
   // UNICODE_TO_GBK[40602] := 16#9A80;
   // UNICODE_TO_GBK[40603] := 16#E6E6;
   // UNICODE_TO_GBK[40604] := 16#9A81;
   // UNICODE_TO_GBK[40605] := 16#E6E7;
   // UNICODE_TO_GBK[40606] := 16#9A82;
   // UNICODE_TO_GBK[40607] := 16#C2EE;
   // UNICODE_TO_GBK[40608] := 16#9A83;
   // UNICODE_TO_GBK[40609] := 16#F353;
   // UNICODE_TO_GBK[40610] := 16#9A84;
   // UNICODE_TO_GBK[40611] := 16#BDBE;
   // UNICODE_TO_GBK[40612] := 16#9A85;
   // UNICODE_TO_GBK[40613] := 16#E6E8;
   // UNICODE_TO_GBK[40614] := 16#9A86;
   // UNICODE_TO_GBK[40615] := 16#C2E6;
   // UNICODE_TO_GBK[40616] := 16#9A87;
   // UNICODE_TO_GBK[40617] := 16#BAA7;
   // UNICODE_TO_GBK[40618] := 16#9A88;
   // UNICODE_TO_GBK[40619] := 16#E6E9;
   // UNICODE_TO_GBK[40620] := 16#9A89;
   // UNICODE_TO_GBK[40621] := 16#F354;
   // UNICODE_TO_GBK[40622] := 16#9A8A;
   // UNICODE_TO_GBK[40623] := 16#E6EA;
   // UNICODE_TO_GBK[40624] := 16#9A8B;
   // UNICODE_TO_GBK[40625] := 16#B3D2;
   // UNICODE_TO_GBK[40626] := 16#9A8C;
   // UNICODE_TO_GBK[40627] := 16#D1E9;
   // UNICODE_TO_GBK[40628] := 16#9A8D;
   // UNICODE_TO_GBK[40629] := 16#F355;
   // UNICODE_TO_GBK[40630] := 16#9A8E;
   // UNICODE_TO_GBK[40631] := 16#F356;
   // UNICODE_TO_GBK[40632] := 16#9A8F;
   // UNICODE_TO_GBK[40633] := 16#BFA5;
   // UNICODE_TO_GBK[40634] := 16#9A90;
   // UNICODE_TO_GBK[40635] := 16#E6EB;
   // UNICODE_TO_GBK[40636] := 16#9A91;
   // UNICODE_TO_GBK[40637] := 16#C6EF;
   // UNICODE_TO_GBK[40638] := 16#9A92;
   // UNICODE_TO_GBK[40639] := 16#E6EC;
   // UNICODE_TO_GBK[40640] := 16#9A93;
   // UNICODE_TO_GBK[40641] := 16#E6ED;
   // UNICODE_TO_GBK[40642] := 16#9A94;
   // UNICODE_TO_GBK[40643] := 16#F357;
   // UNICODE_TO_GBK[40644] := 16#9A95;
   // UNICODE_TO_GBK[40645] := 16#F358;
   // UNICODE_TO_GBK[40646] := 16#9A96;
   // UNICODE_TO_GBK[40647] := 16#E6EE;
   // UNICODE_TO_GBK[40648] := 16#9A97;
   // UNICODE_TO_GBK[40649] := 16#C6AD;
   // UNICODE_TO_GBK[40650] := 16#9A98;
   // UNICODE_TO_GBK[40651] := 16#E6EF;
   // UNICODE_TO_GBK[40652] := 16#9A99;
   // UNICODE_TO_GBK[40653] := 16#F359;
   // UNICODE_TO_GBK[40654] := 16#9A9A;
   // UNICODE_TO_GBK[40655] := 16#C9A7;
   // UNICODE_TO_GBK[40656] := 16#9A9B;
   // UNICODE_TO_GBK[40657] := 16#E6F0;
   // UNICODE_TO_GBK[40658] := 16#9A9C;
   // UNICODE_TO_GBK[40659] := 16#E6F1;
   // UNICODE_TO_GBK[40660] := 16#9A9D;
   // UNICODE_TO_GBK[40661] := 16#E6F2;
   // UNICODE_TO_GBK[40662] := 16#9A9E;
   // UNICODE_TO_GBK[40663] := 16#E5B9;
   // UNICODE_TO_GBK[40664] := 16#9A9F;
   // UNICODE_TO_GBK[40665] := 16#E6F3;
   // UNICODE_TO_GBK[40666] := 16#9AA0;
   // UNICODE_TO_GBK[40667] := 16#E6F4;
   // UNICODE_TO_GBK[40668] := 16#9AA1;
   // UNICODE_TO_GBK[40669] := 16#C2E2;
   // UNICODE_TO_GBK[40670] := 16#9AA2;
   // UNICODE_TO_GBK[40671] := 16#E6F5;
   // UNICODE_TO_GBK[40672] := 16#9AA3;
   // UNICODE_TO_GBK[40673] := 16#E6F6;
   // UNICODE_TO_GBK[40674] := 16#9AA4;
   // UNICODE_TO_GBK[40675] := 16#D6E8;
   // UNICODE_TO_GBK[40676] := 16#9AA5;
   // UNICODE_TO_GBK[40677] := 16#E6F7;
   // UNICODE_TO_GBK[40678] := 16#9AA6;
   // UNICODE_TO_GBK[40679] := 16#F35A;
   // UNICODE_TO_GBK[40680] := 16#9AA7;
   // UNICODE_TO_GBK[40681] := 16#E6F8;
   // UNICODE_TO_GBK[40682] := 16#9AA8;
   // UNICODE_TO_GBK[40683] := 16#B9C7;
   // UNICODE_TO_GBK[40684] := 16#9AA9;
   // UNICODE_TO_GBK[40685] := 16#F35B;
   // UNICODE_TO_GBK[40686] := 16#9AAA;
   // UNICODE_TO_GBK[40687] := 16#F35C;
   // UNICODE_TO_GBK[40688] := 16#9AAB;
   // UNICODE_TO_GBK[40689] := 16#F35D;
   // UNICODE_TO_GBK[40690] := 16#9AAC;
   // UNICODE_TO_GBK[40691] := 16#F35E;
   // UNICODE_TO_GBK[40692] := 16#9AAD;
   // UNICODE_TO_GBK[40693] := 16#F35F;
   // UNICODE_TO_GBK[40694] := 16#9AAE;
   // UNICODE_TO_GBK[40695] := 16#F360;
   // UNICODE_TO_GBK[40696] := 16#9AAF;
   // UNICODE_TO_GBK[40697] := 16#F361;
   // UNICODE_TO_GBK[40698] := 16#9AB0;
   // UNICODE_TO_GBK[40699] := 16#F7BB;
   // UNICODE_TO_GBK[40700] := 16#9AB1;
   // UNICODE_TO_GBK[40701] := 16#F7BA;
   // UNICODE_TO_GBK[40702] := 16#9AB2;
   // UNICODE_TO_GBK[40703] := 16#F362;
   // UNICODE_TO_GBK[40704] := 16#9AB3;
   // UNICODE_TO_GBK[40705] := 16#F363;
   // UNICODE_TO_GBK[40706] := 16#9AB4;
   // UNICODE_TO_GBK[40707] := 16#F364;
   // UNICODE_TO_GBK[40708] := 16#9AB5;
   // UNICODE_TO_GBK[40709] := 16#F365;
   // UNICODE_TO_GBK[40710] := 16#9AB6;
   // UNICODE_TO_GBK[40711] := 16#F7BE;
   // UNICODE_TO_GBK[40712] := 16#9AB7;
   // UNICODE_TO_GBK[40713] := 16#F7BC;
   // UNICODE_TO_GBK[40714] := 16#9AB8;
   // UNICODE_TO_GBK[40715] := 16#BAA1;
   // UNICODE_TO_GBK[40716] := 16#9AB9;
   // UNICODE_TO_GBK[40717] := 16#F366;
   // UNICODE_TO_GBK[40718] := 16#9ABA;
   // UNICODE_TO_GBK[40719] := 16#F7BF;
   // UNICODE_TO_GBK[40720] := 16#9ABB;
   // UNICODE_TO_GBK[40721] := 16#F367;
   // UNICODE_TO_GBK[40722] := 16#9ABC;
   // UNICODE_TO_GBK[40723] := 16#F7C0;
   // UNICODE_TO_GBK[40724] := 16#9ABD;
   // UNICODE_TO_GBK[40725] := 16#F368;
   // UNICODE_TO_GBK[40726] := 16#9ABE;
   // UNICODE_TO_GBK[40727] := 16#F369;
   // UNICODE_TO_GBK[40728] := 16#9ABF;
   // UNICODE_TO_GBK[40729] := 16#F36A;
   // UNICODE_TO_GBK[40730] := 16#9AC0;
   // UNICODE_TO_GBK[40731] := 16#F7C2;
   // UNICODE_TO_GBK[40732] := 16#9AC1;
   // UNICODE_TO_GBK[40733] := 16#F7C1;
   // UNICODE_TO_GBK[40734] := 16#9AC2;
   // UNICODE_TO_GBK[40735] := 16#F7C4;
   // UNICODE_TO_GBK[40736] := 16#9AC3;
   // UNICODE_TO_GBK[40737] := 16#F36B;
   // UNICODE_TO_GBK[40738] := 16#9AC4;
   // UNICODE_TO_GBK[40739] := 16#F36C;
   // UNICODE_TO_GBK[40740] := 16#9AC5;
   // UNICODE_TO_GBK[40741] := 16#F7C3;
   // UNICODE_TO_GBK[40742] := 16#9AC6;
   // UNICODE_TO_GBK[40743] := 16#F36D;
   // UNICODE_TO_GBK[40744] := 16#9AC7;
   // UNICODE_TO_GBK[40745] := 16#F36E;
   // UNICODE_TO_GBK[40746] := 16#9AC8;
   // UNICODE_TO_GBK[40747] := 16#F36F;
   // UNICODE_TO_GBK[40748] := 16#9AC9;
   // UNICODE_TO_GBK[40749] := 16#F370;
   // UNICODE_TO_GBK[40750] := 16#9ACA;
   // UNICODE_TO_GBK[40751] := 16#F371;
   // UNICODE_TO_GBK[40752] := 16#9ACB;
   // UNICODE_TO_GBK[40753] := 16#F7C5;
   // UNICODE_TO_GBK[40754] := 16#9ACC;
   // UNICODE_TO_GBK[40755] := 16#F7C6;
   // UNICODE_TO_GBK[40756] := 16#9ACD;
   // UNICODE_TO_GBK[40757] := 16#F372;
   // UNICODE_TO_GBK[40758] := 16#9ACE;
   // UNICODE_TO_GBK[40759] := 16#F373;
   // UNICODE_TO_GBK[40760] := 16#9ACF;
   // UNICODE_TO_GBK[40761] := 16#F374;
   // UNICODE_TO_GBK[40762] := 16#9AD0;
   // UNICODE_TO_GBK[40763] := 16#F375;
   // UNICODE_TO_GBK[40764] := 16#9AD1;
   // UNICODE_TO_GBK[40765] := 16#F7C7;
   // UNICODE_TO_GBK[40766] := 16#9AD2;
   // UNICODE_TO_GBK[40767] := 16#F376;
   // UNICODE_TO_GBK[40768] := 16#9AD3;
   // UNICODE_TO_GBK[40769] := 16#CBE8;
   // UNICODE_TO_GBK[40770] := 16#9AD4;
   // UNICODE_TO_GBK[40771] := 16#F377;
   // UNICODE_TO_GBK[40772] := 16#9AD5;
   // UNICODE_TO_GBK[40773] := 16#F378;
   // UNICODE_TO_GBK[40774] := 16#9AD6;
   // UNICODE_TO_GBK[40775] := 16#F379;
   // UNICODE_TO_GBK[40776] := 16#9AD7;
   // UNICODE_TO_GBK[40777] := 16#F37A;
   // UNICODE_TO_GBK[40778] := 16#9AD8;
   // UNICODE_TO_GBK[40779] := 16#B8DF;
   // UNICODE_TO_GBK[40780] := 16#9AD9;
   // UNICODE_TO_GBK[40781] := 16#F37B;
   // UNICODE_TO_GBK[40782] := 16#9ADA;
   // UNICODE_TO_GBK[40783] := 16#F37C;
   // UNICODE_TO_GBK[40784] := 16#9ADB;
   // UNICODE_TO_GBK[40785] := 16#F37D;
   // UNICODE_TO_GBK[40786] := 16#9ADC;
   // UNICODE_TO_GBK[40787] := 16#F37E;
   // UNICODE_TO_GBK[40788] := 16#9ADD;
   // UNICODE_TO_GBK[40789] := 16#F380;
   // UNICODE_TO_GBK[40790] := 16#9ADE;
   // UNICODE_TO_GBK[40791] := 16#F381;
   // UNICODE_TO_GBK[40792] := 16#9ADF;
   // UNICODE_TO_GBK[40793] := 16#F7D4;
   // UNICODE_TO_GBK[40794] := 16#9AE0;
   // UNICODE_TO_GBK[40795] := 16#F382;
   // UNICODE_TO_GBK[40796] := 16#9AE1;
   // UNICODE_TO_GBK[40797] := 16#F7D5;
   // UNICODE_TO_GBK[40798] := 16#9AE2;
   // UNICODE_TO_GBK[40799] := 16#F383;
   // UNICODE_TO_GBK[40800] := 16#9AE3;
   // UNICODE_TO_GBK[40801] := 16#F384;
   // UNICODE_TO_GBK[40802] := 16#9AE4;
   // UNICODE_TO_GBK[40803] := 16#F385;
   // UNICODE_TO_GBK[40804] := 16#9AE5;
   // UNICODE_TO_GBK[40805] := 16#F386;
   // UNICODE_TO_GBK[40806] := 16#9AE6;
   // UNICODE_TO_GBK[40807] := 16#F7D6;
   // UNICODE_TO_GBK[40808] := 16#9AE7;
   // UNICODE_TO_GBK[40809] := 16#F387;
   // UNICODE_TO_GBK[40810] := 16#9AE8;
   // UNICODE_TO_GBK[40811] := 16#F388;
   // UNICODE_TO_GBK[40812] := 16#9AE9;
   // UNICODE_TO_GBK[40813] := 16#F389;
   // UNICODE_TO_GBK[40814] := 16#9AEA;
   // UNICODE_TO_GBK[40815] := 16#F38A;
   // UNICODE_TO_GBK[40816] := 16#9AEB;
   // UNICODE_TO_GBK[40817] := 16#F7D8;
   // UNICODE_TO_GBK[40818] := 16#9AEC;
   // UNICODE_TO_GBK[40819] := 16#F38B;
   // UNICODE_TO_GBK[40820] := 16#9AED;
   // UNICODE_TO_GBK[40821] := 16#F7DA;
   // UNICODE_TO_GBK[40822] := 16#9AEE;
   // UNICODE_TO_GBK[40823] := 16#F38C;
   // UNICODE_TO_GBK[40824] := 16#9AEF;
   // UNICODE_TO_GBK[40825] := 16#F7D7;
   // UNICODE_TO_GBK[40826] := 16#9AF0;
   // UNICODE_TO_GBK[40827] := 16#F38D;
   // UNICODE_TO_GBK[40828] := 16#9AF1;
   // UNICODE_TO_GBK[40829] := 16#F38E;
   // UNICODE_TO_GBK[40830] := 16#9AF2;
   // UNICODE_TO_GBK[40831] := 16#F38F;
   // UNICODE_TO_GBK[40832] := 16#9AF3;
   // UNICODE_TO_GBK[40833] := 16#F390;
   // UNICODE_TO_GBK[40834] := 16#9AF4;
   // UNICODE_TO_GBK[40835] := 16#F391;
   // UNICODE_TO_GBK[40836] := 16#9AF5;
   // UNICODE_TO_GBK[40837] := 16#F392;
   // UNICODE_TO_GBK[40838] := 16#9AF6;
   // UNICODE_TO_GBK[40839] := 16#F393;
   // UNICODE_TO_GBK[40840] := 16#9AF7;
   // UNICODE_TO_GBK[40841] := 16#F394;
   // UNICODE_TO_GBK[40842] := 16#9AF8;
   // UNICODE_TO_GBK[40843] := 16#F395;
   // UNICODE_TO_GBK[40844] := 16#9AF9;
   // UNICODE_TO_GBK[40845] := 16#F7DB;
   // UNICODE_TO_GBK[40846] := 16#9AFA;
   // UNICODE_TO_GBK[40847] := 16#F396;
   // UNICODE_TO_GBK[40848] := 16#9AFB;
   // UNICODE_TO_GBK[40849] := 16#F7D9;
   // UNICODE_TO_GBK[40850] := 16#9AFC;
   // UNICODE_TO_GBK[40851] := 16#F397;
   // UNICODE_TO_GBK[40852] := 16#9AFD;
   // UNICODE_TO_GBK[40853] := 16#F398;
   // UNICODE_TO_GBK[40854] := 16#9AFE;
   // UNICODE_TO_GBK[40855] := 16#F399;
   // UNICODE_TO_GBK[40856] := 16#9AFF;
   // UNICODE_TO_GBK[40857] := 16#F39A;
   // UNICODE_TO_GBK[40858] := 16#9B00;
   // UNICODE_TO_GBK[40859] := 16#F39B;
   // UNICODE_TO_GBK[40860] := 16#9B01;
   // UNICODE_TO_GBK[40861] := 16#F39C;
   // UNICODE_TO_GBK[40862] := 16#9B02;
   // UNICODE_TO_GBK[40863] := 16#F39D;
   // UNICODE_TO_GBK[40864] := 16#9B03;
   // UNICODE_TO_GBK[40865] := 16#D7D7;
   // UNICODE_TO_GBK[40866] := 16#9B04;
   // UNICODE_TO_GBK[40867] := 16#F39E;
   // UNICODE_TO_GBK[40868] := 16#9B05;
   // UNICODE_TO_GBK[40869] := 16#F39F;
   // UNICODE_TO_GBK[40870] := 16#9B06;
   // UNICODE_TO_GBK[40871] := 16#F3A0;
   // UNICODE_TO_GBK[40872] := 16#9B07;
   // UNICODE_TO_GBK[40873] := 16#F440;
   // UNICODE_TO_GBK[40874] := 16#9B08;
   // UNICODE_TO_GBK[40875] := 16#F7DC;
   // UNICODE_TO_GBK[40876] := 16#9B09;
   // UNICODE_TO_GBK[40877] := 16#F441;
   // UNICODE_TO_GBK[40878] := 16#9B0A;
   // UNICODE_TO_GBK[40879] := 16#F442;
   // UNICODE_TO_GBK[40880] := 16#9B0B;
   // UNICODE_TO_GBK[40881] := 16#F443;
   // UNICODE_TO_GBK[40882] := 16#9B0C;
   // UNICODE_TO_GBK[40883] := 16#F444;
   // UNICODE_TO_GBK[40884] := 16#9B0D;
   // UNICODE_TO_GBK[40885] := 16#F445;
   // UNICODE_TO_GBK[40886] := 16#9B0E;
   // UNICODE_TO_GBK[40887] := 16#F446;
   // UNICODE_TO_GBK[40888] := 16#9B0F;
   // UNICODE_TO_GBK[40889] := 16#F7DD;
   // UNICODE_TO_GBK[40890] := 16#9B10;
   // UNICODE_TO_GBK[40891] := 16#F447;
   // UNICODE_TO_GBK[40892] := 16#9B11;
   // UNICODE_TO_GBK[40893] := 16#F448;
   // UNICODE_TO_GBK[40894] := 16#9B12;
   // UNICODE_TO_GBK[40895] := 16#F449;
   // UNICODE_TO_GBK[40896] := 16#9B13;
   // UNICODE_TO_GBK[40897] := 16#F7DE;
   // UNICODE_TO_GBK[40898] := 16#9B14;
   // UNICODE_TO_GBK[40899] := 16#F44A;
   // UNICODE_TO_GBK[40900] := 16#9B15;
   // UNICODE_TO_GBK[40901] := 16#F44B;
   // UNICODE_TO_GBK[40902] := 16#9B16;
   // UNICODE_TO_GBK[40903] := 16#F44C;
   // UNICODE_TO_GBK[40904] := 16#9B17;
   // UNICODE_TO_GBK[40905] := 16#F44D;
   // UNICODE_TO_GBK[40906] := 16#9B18;
   // UNICODE_TO_GBK[40907] := 16#F44E;
   // UNICODE_TO_GBK[40908] := 16#9B19;
   // UNICODE_TO_GBK[40909] := 16#F44F;
   // UNICODE_TO_GBK[40910] := 16#9B1A;
   // UNICODE_TO_GBK[40911] := 16#F450;
   // UNICODE_TO_GBK[40912] := 16#9B1B;
   // UNICODE_TO_GBK[40913] := 16#F451;
   // UNICODE_TO_GBK[40914] := 16#9B1C;
   // UNICODE_TO_GBK[40915] := 16#F452;
   // UNICODE_TO_GBK[40916] := 16#9B1D;
   // UNICODE_TO_GBK[40917] := 16#F453;
   // UNICODE_TO_GBK[40918] := 16#9B1E;
   // UNICODE_TO_GBK[40919] := 16#F454;
   // UNICODE_TO_GBK[40920] := 16#9B1F;
   // UNICODE_TO_GBK[40921] := 16#F7DF;
   // UNICODE_TO_GBK[40922] := 16#9B20;
   // UNICODE_TO_GBK[40923] := 16#F455;
   // UNICODE_TO_GBK[40924] := 16#9B21;
   // UNICODE_TO_GBK[40925] := 16#F456;
   // UNICODE_TO_GBK[40926] := 16#9B22;
   // UNICODE_TO_GBK[40927] := 16#F457;
   // UNICODE_TO_GBK[40928] := 16#9B23;
   // UNICODE_TO_GBK[40929] := 16#F7E0;
   // UNICODE_TO_GBK[40930] := 16#9B24;
   // UNICODE_TO_GBK[40931] := 16#F458;
   // UNICODE_TO_GBK[40932] := 16#9B25;
   // UNICODE_TO_GBK[40933] := 16#F459;
   // UNICODE_TO_GBK[40934] := 16#9B26;
   // UNICODE_TO_GBK[40935] := 16#F45A;
   // UNICODE_TO_GBK[40936] := 16#9B27;
   // UNICODE_TO_GBK[40937] := 16#F45B;
   // UNICODE_TO_GBK[40938] := 16#9B28;
   // UNICODE_TO_GBK[40939] := 16#F45C;
   // UNICODE_TO_GBK[40940] := 16#9B29;
   // UNICODE_TO_GBK[40941] := 16#F45D;
   // UNICODE_TO_GBK[40942] := 16#9B2A;
   // UNICODE_TO_GBK[40943] := 16#F45E;
   // UNICODE_TO_GBK[40944] := 16#9B2B;
   // UNICODE_TO_GBK[40945] := 16#F45F;
   // UNICODE_TO_GBK[40946] := 16#9B2C;
   // UNICODE_TO_GBK[40947] := 16#F460;
   // UNICODE_TO_GBK[40948] := 16#9B2D;
   // UNICODE_TO_GBK[40949] := 16#F461;
   // UNICODE_TO_GBK[40950] := 16#9B2E;
   // UNICODE_TO_GBK[40951] := 16#F462;
   // UNICODE_TO_GBK[40952] := 16#9B2F;
   // UNICODE_TO_GBK[40953] := 16#DBCB;
   // UNICODE_TO_GBK[40954] := 16#9B30;
   // UNICODE_TO_GBK[40955] := 16#F463;
   // UNICODE_TO_GBK[40956] := 16#9B31;
   // UNICODE_TO_GBK[40957] := 16#F464;
   // UNICODE_TO_GBK[40958] := 16#9B32;
   // UNICODE_TO_GBK[40959] := 16#D8AA;
   // UNICODE_TO_GBK[40960] := 16#9B33;
   // UNICODE_TO_GBK[40961] := 16#F465;
   // UNICODE_TO_GBK[40962] := 16#9B34;
   // UNICODE_TO_GBK[40963] := 16#F466;
   // UNICODE_TO_GBK[40964] := 16#9B35;
   // UNICODE_TO_GBK[40965] := 16#F467;
   // UNICODE_TO_GBK[40966] := 16#9B36;
   // UNICODE_TO_GBK[40967] := 16#F468;
   // UNICODE_TO_GBK[40968] := 16#9B37;
   // UNICODE_TO_GBK[40969] := 16#F469;
   // UNICODE_TO_GBK[40970] := 16#9B38;
   // UNICODE_TO_GBK[40971] := 16#F46A;
   // UNICODE_TO_GBK[40972] := 16#9B39;
   // UNICODE_TO_GBK[40973] := 16#F46B;
   // UNICODE_TO_GBK[40974] := 16#9B3A;
   // UNICODE_TO_GBK[40975] := 16#F46C;
   // UNICODE_TO_GBK[40976] := 16#9B3B;
   // UNICODE_TO_GBK[40977] := 16#E5F7;
   // UNICODE_TO_GBK[40978] := 16#9B3C;
   // UNICODE_TO_GBK[40979] := 16#B9ED;
   // UNICODE_TO_GBK[40980] := 16#9B3D;
   // UNICODE_TO_GBK[40981] := 16#F46D;
   // UNICODE_TO_GBK[40982] := 16#9B3E;
   // UNICODE_TO_GBK[40983] := 16#F46E;
   // UNICODE_TO_GBK[40984] := 16#9B3F;
   // UNICODE_TO_GBK[40985] := 16#F46F;
   // UNICODE_TO_GBK[40986] := 16#9B40;
   // UNICODE_TO_GBK[40987] := 16#F470;
   // UNICODE_TO_GBK[40988] := 16#9B41;
   // UNICODE_TO_GBK[40989] := 16#BFFD;
   // UNICODE_TO_GBK[40990] := 16#9B42;
   // UNICODE_TO_GBK[40991] := 16#BBEA;
   // UNICODE_TO_GBK[40992] := 16#9B43;
   // UNICODE_TO_GBK[40993] := 16#F7C9;
   // UNICODE_TO_GBK[40994] := 16#9B44;
   // UNICODE_TO_GBK[40995] := 16#C6C7;
   // UNICODE_TO_GBK[40996] := 16#9B45;
   // UNICODE_TO_GBK[40997] := 16#F7C8;
   // UNICODE_TO_GBK[40998] := 16#9B46;
   // UNICODE_TO_GBK[40999] := 16#F471;
   // UNICODE_TO_GBK[41000] := 16#9B47;
   // UNICODE_TO_GBK[41001] := 16#F7CA;
   // UNICODE_TO_GBK[41002] := 16#9B48;
   // UNICODE_TO_GBK[41003] := 16#F7CC;
   // UNICODE_TO_GBK[41004] := 16#9B49;
   // UNICODE_TO_GBK[41005] := 16#F7CB;
   // UNICODE_TO_GBK[41006] := 16#9B4A;
   // UNICODE_TO_GBK[41007] := 16#F472;
   // UNICODE_TO_GBK[41008] := 16#9B4B;
   // UNICODE_TO_GBK[41009] := 16#F473;
   // UNICODE_TO_GBK[41010] := 16#9B4C;
   // UNICODE_TO_GBK[41011] := 16#F474;
   // UNICODE_TO_GBK[41012] := 16#9B4D;
   // UNICODE_TO_GBK[41013] := 16#F7CD;
   // UNICODE_TO_GBK[41014] := 16#9B4E;
   // UNICODE_TO_GBK[41015] := 16#F475;
   // UNICODE_TO_GBK[41016] := 16#9B4F;
   // UNICODE_TO_GBK[41017] := 16#CEBA;
   // UNICODE_TO_GBK[41018] := 16#9B50;
   // UNICODE_TO_GBK[41019] := 16#F476;
   // UNICODE_TO_GBK[41020] := 16#9B51;
   // UNICODE_TO_GBK[41021] := 16#F7CE;
   // UNICODE_TO_GBK[41022] := 16#9B52;
   // UNICODE_TO_GBK[41023] := 16#F477;
   // UNICODE_TO_GBK[41024] := 16#9B53;
   // UNICODE_TO_GBK[41025] := 16#F478;
   // UNICODE_TO_GBK[41026] := 16#9B54;
   // UNICODE_TO_GBK[41027] := 16#C4A7;
   // UNICODE_TO_GBK[41028] := 16#9B55;
   // UNICODE_TO_GBK[41029] := 16#F479;
   // UNICODE_TO_GBK[41030] := 16#9B56;
   // UNICODE_TO_GBK[41031] := 16#F47A;
   // UNICODE_TO_GBK[41032] := 16#9B57;
   // UNICODE_TO_GBK[41033] := 16#F47B;
   // UNICODE_TO_GBK[41034] := 16#9B58;
   // UNICODE_TO_GBK[41035] := 16#F47C;
   // UNICODE_TO_GBK[41036] := 16#9B59;
   // UNICODE_TO_GBK[41037] := 16#F47D;
   // UNICODE_TO_GBK[41038] := 16#9B5A;
   // UNICODE_TO_GBK[41039] := 16#F47E;
   // UNICODE_TO_GBK[41040] := 16#9B5B;
   // UNICODE_TO_GBK[41041] := 16#F480;
   // UNICODE_TO_GBK[41042] := 16#9B5C;
   // UNICODE_TO_GBK[41043] := 16#F481;
   // UNICODE_TO_GBK[41044] := 16#9B5D;
   // UNICODE_TO_GBK[41045] := 16#F482;
   // UNICODE_TO_GBK[41046] := 16#9B5E;
   // UNICODE_TO_GBK[41047] := 16#F483;
   // UNICODE_TO_GBK[41048] := 16#9B5F;
   // UNICODE_TO_GBK[41049] := 16#F484;
   // UNICODE_TO_GBK[41050] := 16#9B60;
   // UNICODE_TO_GBK[41051] := 16#F485;
   // UNICODE_TO_GBK[41052] := 16#9B61;
   // UNICODE_TO_GBK[41053] := 16#F486;
   // UNICODE_TO_GBK[41054] := 16#9B62;
   // UNICODE_TO_GBK[41055] := 16#F487;
   // UNICODE_TO_GBK[41056] := 16#9B63;
   // UNICODE_TO_GBK[41057] := 16#F488;
   // UNICODE_TO_GBK[41058] := 16#9B64;
   // UNICODE_TO_GBK[41059] := 16#F489;
   // UNICODE_TO_GBK[41060] := 16#9B65;
   // UNICODE_TO_GBK[41061] := 16#F48A;
   // UNICODE_TO_GBK[41062] := 16#9B66;
   // UNICODE_TO_GBK[41063] := 16#F48B;
   // UNICODE_TO_GBK[41064] := 16#9B67;
   // UNICODE_TO_GBK[41065] := 16#F48C;
   // UNICODE_TO_GBK[41066] := 16#9B68;
   // UNICODE_TO_GBK[41067] := 16#F48D;
   // UNICODE_TO_GBK[41068] := 16#9B69;
   // UNICODE_TO_GBK[41069] := 16#F48E;
   // UNICODE_TO_GBK[41070] := 16#9B6A;
   // UNICODE_TO_GBK[41071] := 16#F48F;
   // UNICODE_TO_GBK[41072] := 16#9B6B;
   // UNICODE_TO_GBK[41073] := 16#F490;
   // UNICODE_TO_GBK[41074] := 16#9B6C;
   // UNICODE_TO_GBK[41075] := 16#F491;
   // UNICODE_TO_GBK[41076] := 16#9B6D;
   // UNICODE_TO_GBK[41077] := 16#F492;
   // UNICODE_TO_GBK[41078] := 16#9B6E;
   // UNICODE_TO_GBK[41079] := 16#F493;
   // UNICODE_TO_GBK[41080] := 16#9B6F;
   // UNICODE_TO_GBK[41081] := 16#F494;
   // UNICODE_TO_GBK[41082] := 16#9B70;
   // UNICODE_TO_GBK[41083] := 16#F495;
   // UNICODE_TO_GBK[41084] := 16#9B71;
   // UNICODE_TO_GBK[41085] := 16#F496;
   // UNICODE_TO_GBK[41086] := 16#9B72;
   // UNICODE_TO_GBK[41087] := 16#F497;
   // UNICODE_TO_GBK[41088] := 16#9B73;
   // UNICODE_TO_GBK[41089] := 16#F498;
   // UNICODE_TO_GBK[41090] := 16#9B74;
   // UNICODE_TO_GBK[41091] := 16#F499;
   // UNICODE_TO_GBK[41092] := 16#9B75;
   // UNICODE_TO_GBK[41093] := 16#F49A;
   // UNICODE_TO_GBK[41094] := 16#9B76;
   // UNICODE_TO_GBK[41095] := 16#F49B;
   // UNICODE_TO_GBK[41096] := 16#9B77;
   // UNICODE_TO_GBK[41097] := 16#F49C;
   // UNICODE_TO_GBK[41098] := 16#9B78;
   // UNICODE_TO_GBK[41099] := 16#F49D;
   // UNICODE_TO_GBK[41100] := 16#9B79;
   // UNICODE_TO_GBK[41101] := 16#F49E;
   // UNICODE_TO_GBK[41102] := 16#9B7A;
   // UNICODE_TO_GBK[41103] := 16#F49F;
   // UNICODE_TO_GBK[41104] := 16#9B7B;
   // UNICODE_TO_GBK[41105] := 16#F4A0;
   // UNICODE_TO_GBK[41106] := 16#9B7C;
   // UNICODE_TO_GBK[41107] := 16#F540;
   // UNICODE_TO_GBK[41108] := 16#9B7D;
   // UNICODE_TO_GBK[41109] := 16#F541;
   // UNICODE_TO_GBK[41110] := 16#9B7E;
   // UNICODE_TO_GBK[41111] := 16#F542;
   // UNICODE_TO_GBK[41112] := 16#9B7F;
   // UNICODE_TO_GBK[41113] := 16#F543;
   // UNICODE_TO_GBK[41114] := 16#9B80;
   // UNICODE_TO_GBK[41115] := 16#F544;
   // UNICODE_TO_GBK[41116] := 16#9B81;
   // UNICODE_TO_GBK[41117] := 16#F545;
   // UNICODE_TO_GBK[41118] := 16#9B82;
   // UNICODE_TO_GBK[41119] := 16#F546;
   // UNICODE_TO_GBK[41120] := 16#9B83;
   // UNICODE_TO_GBK[41121] := 16#F547;
   // UNICODE_TO_GBK[41122] := 16#9B84;
   // UNICODE_TO_GBK[41123] := 16#F548;
   // UNICODE_TO_GBK[41124] := 16#9B85;
   // UNICODE_TO_GBK[41125] := 16#F549;
   // UNICODE_TO_GBK[41126] := 16#9B86;
   // UNICODE_TO_GBK[41127] := 16#F54A;
   // UNICODE_TO_GBK[41128] := 16#9B87;
   // UNICODE_TO_GBK[41129] := 16#F54B;
   // UNICODE_TO_GBK[41130] := 16#9B88;
   // UNICODE_TO_GBK[41131] := 16#F54C;
   // UNICODE_TO_GBK[41132] := 16#9B89;
   // UNICODE_TO_GBK[41133] := 16#F54D;
   // UNICODE_TO_GBK[41134] := 16#9B8A;
   // UNICODE_TO_GBK[41135] := 16#F54E;
   // UNICODE_TO_GBK[41136] := 16#9B8B;
   // UNICODE_TO_GBK[41137] := 16#F54F;
   // UNICODE_TO_GBK[41138] := 16#9B8C;
   // UNICODE_TO_GBK[41139] := 16#F550;
   // UNICODE_TO_GBK[41140] := 16#9B8D;
   // UNICODE_TO_GBK[41141] := 16#F551;
   // UNICODE_TO_GBK[41142] := 16#9B8E;
   // UNICODE_TO_GBK[41143] := 16#F552;
   // UNICODE_TO_GBK[41144] := 16#9B8F;
   // UNICODE_TO_GBK[41145] := 16#F553;
   // UNICODE_TO_GBK[41146] := 16#9B90;
   // UNICODE_TO_GBK[41147] := 16#F554;
   // UNICODE_TO_GBK[41148] := 16#9B91;
   // UNICODE_TO_GBK[41149] := 16#F555;
   // UNICODE_TO_GBK[41150] := 16#9B92;
   // UNICODE_TO_GBK[41151] := 16#F556;
   // UNICODE_TO_GBK[41152] := 16#9B93;
   // UNICODE_TO_GBK[41153] := 16#F557;
   // UNICODE_TO_GBK[41154] := 16#9B94;
   // UNICODE_TO_GBK[41155] := 16#F558;
   // UNICODE_TO_GBK[41156] := 16#9B95;
   // UNICODE_TO_GBK[41157] := 16#F559;
   // UNICODE_TO_GBK[41158] := 16#9B96;
   // UNICODE_TO_GBK[41159] := 16#F55A;
   // UNICODE_TO_GBK[41160] := 16#9B97;
   // UNICODE_TO_GBK[41161] := 16#F55B;
   // UNICODE_TO_GBK[41162] := 16#9B98;
   // UNICODE_TO_GBK[41163] := 16#F55C;
   // UNICODE_TO_GBK[41164] := 16#9B99;
   // UNICODE_TO_GBK[41165] := 16#F55D;
   // UNICODE_TO_GBK[41166] := 16#9B9A;
   // UNICODE_TO_GBK[41167] := 16#F55E;
   // UNICODE_TO_GBK[41168] := 16#9B9B;
   // UNICODE_TO_GBK[41169] := 16#F55F;
   // UNICODE_TO_GBK[41170] := 16#9B9C;
   // UNICODE_TO_GBK[41171] := 16#F560;
   // UNICODE_TO_GBK[41172] := 16#9B9D;
   // UNICODE_TO_GBK[41173] := 16#F561;
   // UNICODE_TO_GBK[41174] := 16#9B9E;
   // UNICODE_TO_GBK[41175] := 16#F562;
   // UNICODE_TO_GBK[41176] := 16#9B9F;
   // UNICODE_TO_GBK[41177] := 16#F563;
   // UNICODE_TO_GBK[41178] := 16#9BA0;
   // UNICODE_TO_GBK[41179] := 16#F564;
   // UNICODE_TO_GBK[41180] := 16#9BA1;
   // UNICODE_TO_GBK[41181] := 16#F565;
   // UNICODE_TO_GBK[41182] := 16#9BA2;
   // UNICODE_TO_GBK[41183] := 16#F566;
   // UNICODE_TO_GBK[41184] := 16#9BA3;
   // UNICODE_TO_GBK[41185] := 16#F567;
   // UNICODE_TO_GBK[41186] := 16#9BA4;
   // UNICODE_TO_GBK[41187] := 16#F568;
   // UNICODE_TO_GBK[41188] := 16#9BA5;
   // UNICODE_TO_GBK[41189] := 16#F569;
   // UNICODE_TO_GBK[41190] := 16#9BA6;
   // UNICODE_TO_GBK[41191] := 16#F56A;
   // UNICODE_TO_GBK[41192] := 16#9BA7;
   // UNICODE_TO_GBK[41193] := 16#F56B;
   // UNICODE_TO_GBK[41194] := 16#9BA8;
   // UNICODE_TO_GBK[41195] := 16#F56C;
   // UNICODE_TO_GBK[41196] := 16#9BA9;
   // UNICODE_TO_GBK[41197] := 16#F56D;
   // UNICODE_TO_GBK[41198] := 16#9BAA;
   // UNICODE_TO_GBK[41199] := 16#F56E;
   // UNICODE_TO_GBK[41200] := 16#9BAB;
   // UNICODE_TO_GBK[41201] := 16#F56F;
   // UNICODE_TO_GBK[41202] := 16#9BAC;
   // UNICODE_TO_GBK[41203] := 16#F570;
   // UNICODE_TO_GBK[41204] := 16#9BAD;
   // UNICODE_TO_GBK[41205] := 16#F571;
   // UNICODE_TO_GBK[41206] := 16#9BAE;
   // UNICODE_TO_GBK[41207] := 16#F572;
   // UNICODE_TO_GBK[41208] := 16#9BAF;
   // UNICODE_TO_GBK[41209] := 16#F573;
   // UNICODE_TO_GBK[41210] := 16#9BB0;
   // UNICODE_TO_GBK[41211] := 16#F574;
   // UNICODE_TO_GBK[41212] := 16#9BB1;
   // UNICODE_TO_GBK[41213] := 16#F575;
   // UNICODE_TO_GBK[41214] := 16#9BB2;
   // UNICODE_TO_GBK[41215] := 16#F576;
   // UNICODE_TO_GBK[41216] := 16#9BB3;
   // UNICODE_TO_GBK[41217] := 16#F577;
   // UNICODE_TO_GBK[41218] := 16#9BB4;
   // UNICODE_TO_GBK[41219] := 16#F578;
   // UNICODE_TO_GBK[41220] := 16#9BB5;
   // UNICODE_TO_GBK[41221] := 16#F579;
   // UNICODE_TO_GBK[41222] := 16#9BB6;
   // UNICODE_TO_GBK[41223] := 16#F57A;
   // UNICODE_TO_GBK[41224] := 16#9BB7;
   // UNICODE_TO_GBK[41225] := 16#F57B;
   // UNICODE_TO_GBK[41226] := 16#9BB8;
   // UNICODE_TO_GBK[41227] := 16#F57C;
   // UNICODE_TO_GBK[41228] := 16#9BB9;
   // UNICODE_TO_GBK[41229] := 16#F57D;
   // UNICODE_TO_GBK[41230] := 16#9BBA;
   // UNICODE_TO_GBK[41231] := 16#F57E;
   // UNICODE_TO_GBK[41232] := 16#9BBB;
   // UNICODE_TO_GBK[41233] := 16#F580;
   // UNICODE_TO_GBK[41234] := 16#9BBC;
   // UNICODE_TO_GBK[41235] := 16#F581;
   // UNICODE_TO_GBK[41236] := 16#9BBD;
   // UNICODE_TO_GBK[41237] := 16#F582;
   // UNICODE_TO_GBK[41238] := 16#9BBE;
   // UNICODE_TO_GBK[41239] := 16#F583;
   // UNICODE_TO_GBK[41240] := 16#9BBF;
   // UNICODE_TO_GBK[41241] := 16#F584;
   // UNICODE_TO_GBK[41242] := 16#9BC0;
   // UNICODE_TO_GBK[41243] := 16#F585;
   // UNICODE_TO_GBK[41244] := 16#9BC1;
   // UNICODE_TO_GBK[41245] := 16#F586;
   // UNICODE_TO_GBK[41246] := 16#9BC2;
   // UNICODE_TO_GBK[41247] := 16#F587;
   // UNICODE_TO_GBK[41248] := 16#9BC3;
   // UNICODE_TO_GBK[41249] := 16#F588;
   // UNICODE_TO_GBK[41250] := 16#9BC4;
   // UNICODE_TO_GBK[41251] := 16#F589;
   // UNICODE_TO_GBK[41252] := 16#9BC5;
   // UNICODE_TO_GBK[41253] := 16#F58A;
   // UNICODE_TO_GBK[41254] := 16#9BC6;
   // UNICODE_TO_GBK[41255] := 16#F58B;
   // UNICODE_TO_GBK[41256] := 16#9BC7;
   // UNICODE_TO_GBK[41257] := 16#F58C;
   // UNICODE_TO_GBK[41258] := 16#9BC8;
   // UNICODE_TO_GBK[41259] := 16#F58D;
   // UNICODE_TO_GBK[41260] := 16#9BC9;
   // UNICODE_TO_GBK[41261] := 16#F58E;
   // UNICODE_TO_GBK[41262] := 16#9BCA;
   // UNICODE_TO_GBK[41263] := 16#F58F;
   // UNICODE_TO_GBK[41264] := 16#9BCB;
   // UNICODE_TO_GBK[41265] := 16#F590;
   // UNICODE_TO_GBK[41266] := 16#9BCC;
   // UNICODE_TO_GBK[41267] := 16#F591;
   // UNICODE_TO_GBK[41268] := 16#9BCD;
   // UNICODE_TO_GBK[41269] := 16#F592;
   // UNICODE_TO_GBK[41270] := 16#9BCE;
   // UNICODE_TO_GBK[41271] := 16#F593;
   // UNICODE_TO_GBK[41272] := 16#9BCF;
   // UNICODE_TO_GBK[41273] := 16#F594;
   // UNICODE_TO_GBK[41274] := 16#9BD0;
   // UNICODE_TO_GBK[41275] := 16#F595;
   // UNICODE_TO_GBK[41276] := 16#9BD1;
   // UNICODE_TO_GBK[41277] := 16#F596;
   // UNICODE_TO_GBK[41278] := 16#9BD2;
   // UNICODE_TO_GBK[41279] := 16#F597;
   // UNICODE_TO_GBK[41280] := 16#9BD3;
   // UNICODE_TO_GBK[41281] := 16#F598;
   // UNICODE_TO_GBK[41282] := 16#9BD4;
   // UNICODE_TO_GBK[41283] := 16#F599;
   // UNICODE_TO_GBK[41284] := 16#9BD5;
   // UNICODE_TO_GBK[41285] := 16#F59A;
   // UNICODE_TO_GBK[41286] := 16#9BD6;
   // UNICODE_TO_GBK[41287] := 16#F59B;
   // UNICODE_TO_GBK[41288] := 16#9BD7;
   // UNICODE_TO_GBK[41289] := 16#F59C;
   // UNICODE_TO_GBK[41290] := 16#9BD8;
   // UNICODE_TO_GBK[41291] := 16#F59D;
   // UNICODE_TO_GBK[41292] := 16#9BD9;
   // UNICODE_TO_GBK[41293] := 16#F59E;
   // UNICODE_TO_GBK[41294] := 16#9BDA;
   // UNICODE_TO_GBK[41295] := 16#F59F;
   // UNICODE_TO_GBK[41296] := 16#9BDB;
   // UNICODE_TO_GBK[41297] := 16#F5A0;
   // UNICODE_TO_GBK[41298] := 16#9BDC;
   // UNICODE_TO_GBK[41299] := 16#F640;
   // UNICODE_TO_GBK[41300] := 16#9BDD;
   // UNICODE_TO_GBK[41301] := 16#F641;
   // UNICODE_TO_GBK[41302] := 16#9BDE;
   // UNICODE_TO_GBK[41303] := 16#F642;
   // UNICODE_TO_GBK[41304] := 16#9BDF;
   // UNICODE_TO_GBK[41305] := 16#F643;
   // UNICODE_TO_GBK[41306] := 16#9BE0;
   // UNICODE_TO_GBK[41307] := 16#F644;
   // UNICODE_TO_GBK[41308] := 16#9BE1;
   // UNICODE_TO_GBK[41309] := 16#F645;
   // UNICODE_TO_GBK[41310] := 16#9BE2;
   // UNICODE_TO_GBK[41311] := 16#F646;
   // UNICODE_TO_GBK[41312] := 16#9BE3;
   // UNICODE_TO_GBK[41313] := 16#F647;
   // UNICODE_TO_GBK[41314] := 16#9BE4;
   // UNICODE_TO_GBK[41315] := 16#F648;
   // UNICODE_TO_GBK[41316] := 16#9BE5;
   // UNICODE_TO_GBK[41317] := 16#F649;
   // UNICODE_TO_GBK[41318] := 16#9BE6;
   // UNICODE_TO_GBK[41319] := 16#F64A;
   // UNICODE_TO_GBK[41320] := 16#9BE7;
   // UNICODE_TO_GBK[41321] := 16#F64B;
   // UNICODE_TO_GBK[41322] := 16#9BE8;
   // UNICODE_TO_GBK[41323] := 16#F64C;
   // UNICODE_TO_GBK[41324] := 16#9BE9;
   // UNICODE_TO_GBK[41325] := 16#F64D;
   // UNICODE_TO_GBK[41326] := 16#9BEA;
   // UNICODE_TO_GBK[41327] := 16#F64E;
   // UNICODE_TO_GBK[41328] := 16#9BEB;
   // UNICODE_TO_GBK[41329] := 16#F64F;
   // UNICODE_TO_GBK[41330] := 16#9BEC;
   // UNICODE_TO_GBK[41331] := 16#F650;
   // UNICODE_TO_GBK[41332] := 16#9BED;
   // UNICODE_TO_GBK[41333] := 16#F651;
   // UNICODE_TO_GBK[41334] := 16#9BEE;
   // UNICODE_TO_GBK[41335] := 16#F652;
   // UNICODE_TO_GBK[41336] := 16#9BEF;
   // UNICODE_TO_GBK[41337] := 16#F653;
   // UNICODE_TO_GBK[41338] := 16#9BF0;
   // UNICODE_TO_GBK[41339] := 16#F654;
   // UNICODE_TO_GBK[41340] := 16#9BF1;
   // UNICODE_TO_GBK[41341] := 16#F655;
   // UNICODE_TO_GBK[41342] := 16#9BF2;
   // UNICODE_TO_GBK[41343] := 16#F656;
   // UNICODE_TO_GBK[41344] := 16#9BF3;
   // UNICODE_TO_GBK[41345] := 16#F657;
   // UNICODE_TO_GBK[41346] := 16#9BF4;
   // UNICODE_TO_GBK[41347] := 16#F658;
   // UNICODE_TO_GBK[41348] := 16#9BF5;
   // UNICODE_TO_GBK[41349] := 16#F659;
   // UNICODE_TO_GBK[41350] := 16#9BF6;
   // UNICODE_TO_GBK[41351] := 16#F65A;
   // UNICODE_TO_GBK[41352] := 16#9BF7;
   // UNICODE_TO_GBK[41353] := 16#F65B;
   // UNICODE_TO_GBK[41354] := 16#9BF8;
   // UNICODE_TO_GBK[41355] := 16#F65C;
   // UNICODE_TO_GBK[41356] := 16#9BF9;
   // UNICODE_TO_GBK[41357] := 16#F65D;
   // UNICODE_TO_GBK[41358] := 16#9BFA;
   // UNICODE_TO_GBK[41359] := 16#F65E;
   // UNICODE_TO_GBK[41360] := 16#9BFB;
   // UNICODE_TO_GBK[41361] := 16#F65F;
   // UNICODE_TO_GBK[41362] := 16#9BFC;
   // UNICODE_TO_GBK[41363] := 16#F660;
   // UNICODE_TO_GBK[41364] := 16#9BFD;
   // UNICODE_TO_GBK[41365] := 16#F661;
   // UNICODE_TO_GBK[41366] := 16#9BFE;
   // UNICODE_TO_GBK[41367] := 16#F662;
   // UNICODE_TO_GBK[41368] := 16#9BFF;
   // UNICODE_TO_GBK[41369] := 16#F663;
   // UNICODE_TO_GBK[41370] := 16#9C00;
   // UNICODE_TO_GBK[41371] := 16#F664;
   // UNICODE_TO_GBK[41372] := 16#9C01;
   // UNICODE_TO_GBK[41373] := 16#F665;
   // UNICODE_TO_GBK[41374] := 16#9C02;
   // UNICODE_TO_GBK[41375] := 16#F666;
   // UNICODE_TO_GBK[41376] := 16#9C03;
   // UNICODE_TO_GBK[41377] := 16#F667;
   // UNICODE_TO_GBK[41378] := 16#9C04;
   // UNICODE_TO_GBK[41379] := 16#F668;
   // UNICODE_TO_GBK[41380] := 16#9C05;
   // UNICODE_TO_GBK[41381] := 16#F669;
   // UNICODE_TO_GBK[41382] := 16#9C06;
   // UNICODE_TO_GBK[41383] := 16#F66A;
   // UNICODE_TO_GBK[41384] := 16#9C07;
   // UNICODE_TO_GBK[41385] := 16#F66B;
   // UNICODE_TO_GBK[41386] := 16#9C08;
   // UNICODE_TO_GBK[41387] := 16#F66C;
   // UNICODE_TO_GBK[41388] := 16#9C09;
   // UNICODE_TO_GBK[41389] := 16#F66D;
   // UNICODE_TO_GBK[41390] := 16#9C0A;
   // UNICODE_TO_GBK[41391] := 16#F66E;
   // UNICODE_TO_GBK[41392] := 16#9C0B;
   // UNICODE_TO_GBK[41393] := 16#F66F;
   // UNICODE_TO_GBK[41394] := 16#9C0C;
   // UNICODE_TO_GBK[41395] := 16#F670;
   // UNICODE_TO_GBK[41396] := 16#9C0D;
   // UNICODE_TO_GBK[41397] := 16#F671;
   // UNICODE_TO_GBK[41398] := 16#9C0E;
   // UNICODE_TO_GBK[41399] := 16#F672;
   // UNICODE_TO_GBK[41400] := 16#9C0F;
   // UNICODE_TO_GBK[41401] := 16#F673;
   // UNICODE_TO_GBK[41402] := 16#9C10;
   // UNICODE_TO_GBK[41403] := 16#F674;
   // UNICODE_TO_GBK[41404] := 16#9C11;
   // UNICODE_TO_GBK[41405] := 16#F675;
   // UNICODE_TO_GBK[41406] := 16#9C12;
   // UNICODE_TO_GBK[41407] := 16#F676;
   // UNICODE_TO_GBK[41408] := 16#9C13;
   // UNICODE_TO_GBK[41409] := 16#F677;
   // UNICODE_TO_GBK[41410] := 16#9C14;
   // UNICODE_TO_GBK[41411] := 16#F678;
   // UNICODE_TO_GBK[41412] := 16#9C15;
   // UNICODE_TO_GBK[41413] := 16#F679;
   // UNICODE_TO_GBK[41414] := 16#9C16;
   // UNICODE_TO_GBK[41415] := 16#F67A;
   // UNICODE_TO_GBK[41416] := 16#9C17;
   // UNICODE_TO_GBK[41417] := 16#F67B;
   // UNICODE_TO_GBK[41418] := 16#9C18;
   // UNICODE_TO_GBK[41419] := 16#F67C;
   // UNICODE_TO_GBK[41420] := 16#9C19;
   // UNICODE_TO_GBK[41421] := 16#F67D;
   // UNICODE_TO_GBK[41422] := 16#9C1A;
   // UNICODE_TO_GBK[41423] := 16#F67E;
   // UNICODE_TO_GBK[41424] := 16#9C1B;
   // UNICODE_TO_GBK[41425] := 16#F680;
   // UNICODE_TO_GBK[41426] := 16#9C1C;
   // UNICODE_TO_GBK[41427] := 16#F681;
   // UNICODE_TO_GBK[41428] := 16#9C1D;
   // UNICODE_TO_GBK[41429] := 16#F682;
   // UNICODE_TO_GBK[41430] := 16#9C1E;
   // UNICODE_TO_GBK[41431] := 16#F683;
   // UNICODE_TO_GBK[41432] := 16#9C1F;
   // UNICODE_TO_GBK[41433] := 16#F684;
   // UNICODE_TO_GBK[41434] := 16#9C20;
   // UNICODE_TO_GBK[41435] := 16#F685;
   // UNICODE_TO_GBK[41436] := 16#9C21;
   // UNICODE_TO_GBK[41437] := 16#F686;
   // UNICODE_TO_GBK[41438] := 16#9C22;
   // UNICODE_TO_GBK[41439] := 16#F687;
   // UNICODE_TO_GBK[41440] := 16#9C23;
   // UNICODE_TO_GBK[41441] := 16#F688;
   // UNICODE_TO_GBK[41442] := 16#9C24;
   // UNICODE_TO_GBK[41443] := 16#F689;
   // UNICODE_TO_GBK[41444] := 16#9C25;
   // UNICODE_TO_GBK[41445] := 16#F68A;
   // UNICODE_TO_GBK[41446] := 16#9C26;
   // UNICODE_TO_GBK[41447] := 16#F68B;
   // UNICODE_TO_GBK[41448] := 16#9C27;
   // UNICODE_TO_GBK[41449] := 16#F68C;
   // UNICODE_TO_GBK[41450] := 16#9C28;
   // UNICODE_TO_GBK[41451] := 16#F68D;
   // UNICODE_TO_GBK[41452] := 16#9C29;
   // UNICODE_TO_GBK[41453] := 16#F68E;
   // UNICODE_TO_GBK[41454] := 16#9C2A;
   // UNICODE_TO_GBK[41455] := 16#F68F;
   // UNICODE_TO_GBK[41456] := 16#9C2B;
   // UNICODE_TO_GBK[41457] := 16#F690;
   // UNICODE_TO_GBK[41458] := 16#9C2C;
   // UNICODE_TO_GBK[41459] := 16#F691;
   // UNICODE_TO_GBK[41460] := 16#9C2D;
   // UNICODE_TO_GBK[41461] := 16#F692;
   // UNICODE_TO_GBK[41462] := 16#9C2E;
   // UNICODE_TO_GBK[41463] := 16#F693;
   // UNICODE_TO_GBK[41464] := 16#9C2F;
   // UNICODE_TO_GBK[41465] := 16#F694;
   // UNICODE_TO_GBK[41466] := 16#9C30;
   // UNICODE_TO_GBK[41467] := 16#F695;
   // UNICODE_TO_GBK[41468] := 16#9C31;
   // UNICODE_TO_GBK[41469] := 16#F696;
   // UNICODE_TO_GBK[41470] := 16#9C32;
   // UNICODE_TO_GBK[41471] := 16#F697;
   // UNICODE_TO_GBK[41472] := 16#9C33;
   // UNICODE_TO_GBK[41473] := 16#F698;
   // UNICODE_TO_GBK[41474] := 16#9C34;
   // UNICODE_TO_GBK[41475] := 16#F699;
   // UNICODE_TO_GBK[41476] := 16#9C35;
   // UNICODE_TO_GBK[41477] := 16#F69A;
   // UNICODE_TO_GBK[41478] := 16#9C36;
   // UNICODE_TO_GBK[41479] := 16#F69B;
   // UNICODE_TO_GBK[41480] := 16#9C37;
   // UNICODE_TO_GBK[41481] := 16#F69C;
   // UNICODE_TO_GBK[41482] := 16#9C38;
   // UNICODE_TO_GBK[41483] := 16#F69D;
   // UNICODE_TO_GBK[41484] := 16#9C39;
   // UNICODE_TO_GBK[41485] := 16#F69E;
   // UNICODE_TO_GBK[41486] := 16#9C3A;
   // UNICODE_TO_GBK[41487] := 16#F69F;
   // UNICODE_TO_GBK[41488] := 16#9C3B;
   // UNICODE_TO_GBK[41489] := 16#F6A0;
   // UNICODE_TO_GBK[41490] := 16#9C3C;
   // UNICODE_TO_GBK[41491] := 16#F740;
   // UNICODE_TO_GBK[41492] := 16#9C3D;
   // UNICODE_TO_GBK[41493] := 16#F741;
   // UNICODE_TO_GBK[41494] := 16#9C3E;
   // UNICODE_TO_GBK[41495] := 16#F742;
   // UNICODE_TO_GBK[41496] := 16#9C3F;
   // UNICODE_TO_GBK[41497] := 16#F743;
   // UNICODE_TO_GBK[41498] := 16#9C40;
   // UNICODE_TO_GBK[41499] := 16#F744;
   // UNICODE_TO_GBK[41500] := 16#9C41;
   // UNICODE_TO_GBK[41501] := 16#F745;
   // UNICODE_TO_GBK[41502] := 16#9C42;
   // UNICODE_TO_GBK[41503] := 16#F746;
   // UNICODE_TO_GBK[41504] := 16#9C43;
   // UNICODE_TO_GBK[41505] := 16#F747;
   // UNICODE_TO_GBK[41506] := 16#9C44;
   // UNICODE_TO_GBK[41507] := 16#F748;
   // UNICODE_TO_GBK[41508] := 16#9C45;
   // UNICODE_TO_GBK[41509] := 16#F749;
   // UNICODE_TO_GBK[41510] := 16#9C46;
   // UNICODE_TO_GBK[41511] := 16#F74A;
   // UNICODE_TO_GBK[41512] := 16#9C47;
   // UNICODE_TO_GBK[41513] := 16#F74B;
   // UNICODE_TO_GBK[41514] := 16#9C48;
   // UNICODE_TO_GBK[41515] := 16#F74C;
   // UNICODE_TO_GBK[41516] := 16#9C49;
   // UNICODE_TO_GBK[41517] := 16#F74D;
   // UNICODE_TO_GBK[41518] := 16#9C4A;
   // UNICODE_TO_GBK[41519] := 16#F74E;
   // UNICODE_TO_GBK[41520] := 16#9C4B;
   // UNICODE_TO_GBK[41521] := 16#F74F;
   // UNICODE_TO_GBK[41522] := 16#9C4C;
   // UNICODE_TO_GBK[41523] := 16#F750;
   // UNICODE_TO_GBK[41524] := 16#9C4D;
   // UNICODE_TO_GBK[41525] := 16#F751;
   // UNICODE_TO_GBK[41526] := 16#9C4E;
   // UNICODE_TO_GBK[41527] := 16#F752;
   // UNICODE_TO_GBK[41528] := 16#9C4F;
   // UNICODE_TO_GBK[41529] := 16#F753;
   // UNICODE_TO_GBK[41530] := 16#9C50;
   // UNICODE_TO_GBK[41531] := 16#F754;
   // UNICODE_TO_GBK[41532] := 16#9C51;
   // UNICODE_TO_GBK[41533] := 16#F755;
   // UNICODE_TO_GBK[41534] := 16#9C52;
   // UNICODE_TO_GBK[41535] := 16#F756;
   // UNICODE_TO_GBK[41536] := 16#9C53;
   // UNICODE_TO_GBK[41537] := 16#F757;
   // UNICODE_TO_GBK[41538] := 16#9C54;
   // UNICODE_TO_GBK[41539] := 16#F758;
   // UNICODE_TO_GBK[41540] := 16#9C55;
   // UNICODE_TO_GBK[41541] := 16#F759;
   // UNICODE_TO_GBK[41542] := 16#9C56;
   // UNICODE_TO_GBK[41543] := 16#F75A;
   // UNICODE_TO_GBK[41544] := 16#9C57;
   // UNICODE_TO_GBK[41545] := 16#F75B;
   // UNICODE_TO_GBK[41546] := 16#9C58;
   // UNICODE_TO_GBK[41547] := 16#F75C;
   // UNICODE_TO_GBK[41548] := 16#9C59;
   // UNICODE_TO_GBK[41549] := 16#F75D;
   // UNICODE_TO_GBK[41550] := 16#9C5A;
   // UNICODE_TO_GBK[41551] := 16#F75E;
   // UNICODE_TO_GBK[41552] := 16#9C5B;
   // UNICODE_TO_GBK[41553] := 16#F75F;
   // UNICODE_TO_GBK[41554] := 16#9C5C;
   // UNICODE_TO_GBK[41555] := 16#F760;
   // UNICODE_TO_GBK[41556] := 16#9C5D;
   // UNICODE_TO_GBK[41557] := 16#F761;
   // UNICODE_TO_GBK[41558] := 16#9C5E;
   // UNICODE_TO_GBK[41559] := 16#F762;
   // UNICODE_TO_GBK[41560] := 16#9C5F;
   // UNICODE_TO_GBK[41561] := 16#F763;
   // UNICODE_TO_GBK[41562] := 16#9C60;
   // UNICODE_TO_GBK[41563] := 16#F764;
   // UNICODE_TO_GBK[41564] := 16#9C61;
   // UNICODE_TO_GBK[41565] := 16#F765;
   // UNICODE_TO_GBK[41566] := 16#9C62;
   // UNICODE_TO_GBK[41567] := 16#F766;
   // UNICODE_TO_GBK[41568] := 16#9C63;
   // UNICODE_TO_GBK[41569] := 16#F767;
   // UNICODE_TO_GBK[41570] := 16#9C64;
   // UNICODE_TO_GBK[41571] := 16#F768;
   // UNICODE_TO_GBK[41572] := 16#9C65;
   // UNICODE_TO_GBK[41573] := 16#F769;
   // UNICODE_TO_GBK[41574] := 16#9C66;
   // UNICODE_TO_GBK[41575] := 16#F76A;
   // UNICODE_TO_GBK[41576] := 16#9C67;
   // UNICODE_TO_GBK[41577] := 16#F76B;
   // UNICODE_TO_GBK[41578] := 16#9C68;
   // UNICODE_TO_GBK[41579] := 16#F76C;
   // UNICODE_TO_GBK[41580] := 16#9C69;
   // UNICODE_TO_GBK[41581] := 16#F76D;
   // UNICODE_TO_GBK[41582] := 16#9C6A;
   // UNICODE_TO_GBK[41583] := 16#F76E;
   // UNICODE_TO_GBK[41584] := 16#9C6B;
   // UNICODE_TO_GBK[41585] := 16#F76F;
   // UNICODE_TO_GBK[41586] := 16#9C6C;
   // UNICODE_TO_GBK[41587] := 16#F770;
   // UNICODE_TO_GBK[41588] := 16#9C6D;
   // UNICODE_TO_GBK[41589] := 16#F771;
   // UNICODE_TO_GBK[41590] := 16#9C6E;
   // UNICODE_TO_GBK[41591] := 16#F772;
   // UNICODE_TO_GBK[41592] := 16#9C6F;
   // UNICODE_TO_GBK[41593] := 16#F773;
   // UNICODE_TO_GBK[41594] := 16#9C70;
   // UNICODE_TO_GBK[41595] := 16#F774;
   // UNICODE_TO_GBK[41596] := 16#9C71;
   // UNICODE_TO_GBK[41597] := 16#F775;
   // UNICODE_TO_GBK[41598] := 16#9C72;
   // UNICODE_TO_GBK[41599] := 16#F776;
   // UNICODE_TO_GBK[41600] := 16#9C73;
   // UNICODE_TO_GBK[41601] := 16#F777;
   // UNICODE_TO_GBK[41602] := 16#9C74;
   // UNICODE_TO_GBK[41603] := 16#F778;
   // UNICODE_TO_GBK[41604] := 16#9C75;
   // UNICODE_TO_GBK[41605] := 16#F779;
   // UNICODE_TO_GBK[41606] := 16#9C76;
   // UNICODE_TO_GBK[41607] := 16#F77A;
   // UNICODE_TO_GBK[41608] := 16#9C77;
   // UNICODE_TO_GBK[41609] := 16#F77B;
   // UNICODE_TO_GBK[41610] := 16#9C78;
   // UNICODE_TO_GBK[41611] := 16#F77C;
   // UNICODE_TO_GBK[41612] := 16#9C79;
   // UNICODE_TO_GBK[41613] := 16#F77D;
   // UNICODE_TO_GBK[41614] := 16#9C7A;
   // UNICODE_TO_GBK[41615] := 16#F77E;
   // UNICODE_TO_GBK[41616] := 16#9C7B;
   // UNICODE_TO_GBK[41617] := 16#F780;
   // UNICODE_TO_GBK[41618] := 16#9C7C;
   // UNICODE_TO_GBK[41619] := 16#D3E3;
   // UNICODE_TO_GBK[41620] := 16#9C7D;
   // UNICODE_TO_GBK[41621] := 16#F781;
   // UNICODE_TO_GBK[41622] := 16#9C7E;
   // UNICODE_TO_GBK[41623] := 16#F782;
   // UNICODE_TO_GBK[41624] := 16#9C7F;
   // UNICODE_TO_GBK[41625] := 16#F6CF;
   // UNICODE_TO_GBK[41626] := 16#9C80;
   // UNICODE_TO_GBK[41627] := 16#F783;
   // UNICODE_TO_GBK[41628] := 16#9C81;
   // UNICODE_TO_GBK[41629] := 16#C2B3;
   // UNICODE_TO_GBK[41630] := 16#9C82;
   // UNICODE_TO_GBK[41631] := 16#F6D0;
   // UNICODE_TO_GBK[41632] := 16#9C83;
   // UNICODE_TO_GBK[41633] := 16#F784;
   // UNICODE_TO_GBK[41634] := 16#9C84;
   // UNICODE_TO_GBK[41635] := 16#F785;
   // UNICODE_TO_GBK[41636] := 16#9C85;
   // UNICODE_TO_GBK[41637] := 16#F6D1;
   // UNICODE_TO_GBK[41638] := 16#9C86;
   // UNICODE_TO_GBK[41639] := 16#F6D2;
   // UNICODE_TO_GBK[41640] := 16#9C87;
   // UNICODE_TO_GBK[41641] := 16#F6D3;
   // UNICODE_TO_GBK[41642] := 16#9C88;
   // UNICODE_TO_GBK[41643] := 16#F6D4;
   // UNICODE_TO_GBK[41644] := 16#9C89;
   // UNICODE_TO_GBK[41645] := 16#F786;
   // UNICODE_TO_GBK[41646] := 16#9C8A;
   // UNICODE_TO_GBK[41647] := 16#F787;
   // UNICODE_TO_GBK[41648] := 16#9C8B;
   // UNICODE_TO_GBK[41649] := 16#F6D6;
   // UNICODE_TO_GBK[41650] := 16#9C8C;
   // UNICODE_TO_GBK[41651] := 16#F788;
   // UNICODE_TO_GBK[41652] := 16#9C8D;
   // UNICODE_TO_GBK[41653] := 16#B1AB;
   // UNICODE_TO_GBK[41654] := 16#9C8E;
   // UNICODE_TO_GBK[41655] := 16#F6D7;
   // UNICODE_TO_GBK[41656] := 16#9C8F;
   // UNICODE_TO_GBK[41657] := 16#F789;
   // UNICODE_TO_GBK[41658] := 16#9C90;
   // UNICODE_TO_GBK[41659] := 16#F6D8;
   // UNICODE_TO_GBK[41660] := 16#9C91;
   // UNICODE_TO_GBK[41661] := 16#F6D9;
   // UNICODE_TO_GBK[41662] := 16#9C92;
   // UNICODE_TO_GBK[41663] := 16#F6DA;
   // UNICODE_TO_GBK[41664] := 16#9C93;
   // UNICODE_TO_GBK[41665] := 16#F78A;
   // UNICODE_TO_GBK[41666] := 16#9C94;
   // UNICODE_TO_GBK[41667] := 16#F6DB;
   // UNICODE_TO_GBK[41668] := 16#9C95;
   // UNICODE_TO_GBK[41669] := 16#F6DC;
   // UNICODE_TO_GBK[41670] := 16#9C96;
   // UNICODE_TO_GBK[41671] := 16#F78B;
   // UNICODE_TO_GBK[41672] := 16#9C97;
   // UNICODE_TO_GBK[41673] := 16#F78C;
   // UNICODE_TO_GBK[41674] := 16#9C98;
   // UNICODE_TO_GBK[41675] := 16#F78D;
   // UNICODE_TO_GBK[41676] := 16#9C99;
   // UNICODE_TO_GBK[41677] := 16#F78E;
   // UNICODE_TO_GBK[41678] := 16#9C9A;
   // UNICODE_TO_GBK[41679] := 16#F6DD;
   // UNICODE_TO_GBK[41680] := 16#9C9B;
   // UNICODE_TO_GBK[41681] := 16#F6DE;
   // UNICODE_TO_GBK[41682] := 16#9C9C;
   // UNICODE_TO_GBK[41683] := 16#CFCA;
   // UNICODE_TO_GBK[41684] := 16#9C9D;
   // UNICODE_TO_GBK[41685] := 16#F78F;
   // UNICODE_TO_GBK[41686] := 16#9C9E;
   // UNICODE_TO_GBK[41687] := 16#F6DF;
   // UNICODE_TO_GBK[41688] := 16#9C9F;
   // UNICODE_TO_GBK[41689] := 16#F6E0;
   // UNICODE_TO_GBK[41690] := 16#9CA0;
   // UNICODE_TO_GBK[41691] := 16#F6E1;
   // UNICODE_TO_GBK[41692] := 16#9CA1;
   // UNICODE_TO_GBK[41693] := 16#F6E2;
   // UNICODE_TO_GBK[41694] := 16#9CA2;
   // UNICODE_TO_GBK[41695] := 16#F6E3;
   // UNICODE_TO_GBK[41696] := 16#9CA3;
   // UNICODE_TO_GBK[41697] := 16#F6E4;
   // UNICODE_TO_GBK[41698] := 16#9CA4;
   // UNICODE_TO_GBK[41699] := 16#C0F0;
   // UNICODE_TO_GBK[41700] := 16#9CA5;
   // UNICODE_TO_GBK[41701] := 16#F6E5;
   // UNICODE_TO_GBK[41702] := 16#9CA6;
   // UNICODE_TO_GBK[41703] := 16#F6E6;
   // UNICODE_TO_GBK[41704] := 16#9CA7;
   // UNICODE_TO_GBK[41705] := 16#F6E7;
   // UNICODE_TO_GBK[41706] := 16#9CA8;
   // UNICODE_TO_GBK[41707] := 16#F6E8;
   // UNICODE_TO_GBK[41708] := 16#9CA9;
   // UNICODE_TO_GBK[41709] := 16#F6E9;
   // UNICODE_TO_GBK[41710] := 16#9CAA;
   // UNICODE_TO_GBK[41711] := 16#F790;
   // UNICODE_TO_GBK[41712] := 16#9CAB;
   // UNICODE_TO_GBK[41713] := 16#F6EA;
   // UNICODE_TO_GBK[41714] := 16#9CAC;
   // UNICODE_TO_GBK[41715] := 16#F791;
   // UNICODE_TO_GBK[41716] := 16#9CAD;
   // UNICODE_TO_GBK[41717] := 16#F6EB;
   // UNICODE_TO_GBK[41718] := 16#9CAE;
   // UNICODE_TO_GBK[41719] := 16#F6EC;
   // UNICODE_TO_GBK[41720] := 16#9CAF;
   // UNICODE_TO_GBK[41721] := 16#F792;
   // UNICODE_TO_GBK[41722] := 16#9CB0;
   // UNICODE_TO_GBK[41723] := 16#F6ED;
   // UNICODE_TO_GBK[41724] := 16#9CB1;
   // UNICODE_TO_GBK[41725] := 16#F6EE;
   // UNICODE_TO_GBK[41726] := 16#9CB2;
   // UNICODE_TO_GBK[41727] := 16#F6EF;
   // UNICODE_TO_GBK[41728] := 16#9CB3;
   // UNICODE_TO_GBK[41729] := 16#F6F0;
   // UNICODE_TO_GBK[41730] := 16#9CB4;
   // UNICODE_TO_GBK[41731] := 16#F6F1;
   // UNICODE_TO_GBK[41732] := 16#9CB5;
   // UNICODE_TO_GBK[41733] := 16#F6F2;
   // UNICODE_TO_GBK[41734] := 16#9CB6;
   // UNICODE_TO_GBK[41735] := 16#F6F3;
   // UNICODE_TO_GBK[41736] := 16#9CB7;
   // UNICODE_TO_GBK[41737] := 16#F6F4;
   // UNICODE_TO_GBK[41738] := 16#9CB8;
   // UNICODE_TO_GBK[41739] := 16#BEA8;
   // UNICODE_TO_GBK[41740] := 16#9CB9;
   // UNICODE_TO_GBK[41741] := 16#F793;
   // UNICODE_TO_GBK[41742] := 16#9CBA;
   // UNICODE_TO_GBK[41743] := 16#F6F5;
   // UNICODE_TO_GBK[41744] := 16#9CBB;
   // UNICODE_TO_GBK[41745] := 16#F6F6;
   // UNICODE_TO_GBK[41746] := 16#9CBC;
   // UNICODE_TO_GBK[41747] := 16#F6F7;
   // UNICODE_TO_GBK[41748] := 16#9CBD;
   // UNICODE_TO_GBK[41749] := 16#F6F8;
   // UNICODE_TO_GBK[41750] := 16#9CBE;
   // UNICODE_TO_GBK[41751] := 16#F794;
   // UNICODE_TO_GBK[41752] := 16#9CBF;
   // UNICODE_TO_GBK[41753] := 16#F795;
   // UNICODE_TO_GBK[41754] := 16#9CC0;
   // UNICODE_TO_GBK[41755] := 16#F796;
   // UNICODE_TO_GBK[41756] := 16#9CC1;
   // UNICODE_TO_GBK[41757] := 16#F797;
   // UNICODE_TO_GBK[41758] := 16#9CC2;
   // UNICODE_TO_GBK[41759] := 16#F798;
   // UNICODE_TO_GBK[41760] := 16#9CC3;
   // UNICODE_TO_GBK[41761] := 16#C8FA;
   // UNICODE_TO_GBK[41762] := 16#9CC4;
   // UNICODE_TO_GBK[41763] := 16#F6F9;
   // UNICODE_TO_GBK[41764] := 16#9CC5;
   // UNICODE_TO_GBK[41765] := 16#F6FA;
   // UNICODE_TO_GBK[41766] := 16#9CC6;
   // UNICODE_TO_GBK[41767] := 16#F6FB;
   // UNICODE_TO_GBK[41768] := 16#9CC7;
   // UNICODE_TO_GBK[41769] := 16#F6FC;
   // UNICODE_TO_GBK[41770] := 16#9CC8;
   // UNICODE_TO_GBK[41771] := 16#F799;
   // UNICODE_TO_GBK[41772] := 16#9CC9;
   // UNICODE_TO_GBK[41773] := 16#F79A;
   // UNICODE_TO_GBK[41774] := 16#9CCA;
   // UNICODE_TO_GBK[41775] := 16#F6FD;
   // UNICODE_TO_GBK[41776] := 16#9CCB;
   // UNICODE_TO_GBK[41777] := 16#F6FE;
   // UNICODE_TO_GBK[41778] := 16#9CCC;
   // UNICODE_TO_GBK[41779] := 16#F7A1;
   // UNICODE_TO_GBK[41780] := 16#9CCD;
   // UNICODE_TO_GBK[41781] := 16#F7A2;
   // UNICODE_TO_GBK[41782] := 16#9CCE;
   // UNICODE_TO_GBK[41783] := 16#F7A3;
   // UNICODE_TO_GBK[41784] := 16#9CCF;
   // UNICODE_TO_GBK[41785] := 16#F7A4;
   // UNICODE_TO_GBK[41786] := 16#9CD0;
   // UNICODE_TO_GBK[41787] := 16#F7A5;
   // UNICODE_TO_GBK[41788] := 16#9CD1;
   // UNICODE_TO_GBK[41789] := 16#F79B;
   // UNICODE_TO_GBK[41790] := 16#9CD2;
   // UNICODE_TO_GBK[41791] := 16#F79C;
   // UNICODE_TO_GBK[41792] := 16#9CD3;
   // UNICODE_TO_GBK[41793] := 16#F7A6;
   // UNICODE_TO_GBK[41794] := 16#9CD4;
   // UNICODE_TO_GBK[41795] := 16#F7A7;
   // UNICODE_TO_GBK[41796] := 16#9CD5;
   // UNICODE_TO_GBK[41797] := 16#F7A8;
   // UNICODE_TO_GBK[41798] := 16#9CD6;
   // UNICODE_TO_GBK[41799] := 16#B1EE;
   // UNICODE_TO_GBK[41800] := 16#9CD7;
   // UNICODE_TO_GBK[41801] := 16#F7A9;
   // UNICODE_TO_GBK[41802] := 16#9CD8;
   // UNICODE_TO_GBK[41803] := 16#F7AA;
   // UNICODE_TO_GBK[41804] := 16#9CD9;
   // UNICODE_TO_GBK[41805] := 16#F7AB;
   // UNICODE_TO_GBK[41806] := 16#9CDA;
   // UNICODE_TO_GBK[41807] := 16#F79D;
   // UNICODE_TO_GBK[41808] := 16#9CDB;
   // UNICODE_TO_GBK[41809] := 16#F79E;
   // UNICODE_TO_GBK[41810] := 16#9CDC;
   // UNICODE_TO_GBK[41811] := 16#F7AC;
   // UNICODE_TO_GBK[41812] := 16#9CDD;
   // UNICODE_TO_GBK[41813] := 16#F7AD;
   // UNICODE_TO_GBK[41814] := 16#9CDE;
   // UNICODE_TO_GBK[41815] := 16#C1DB;
   // UNICODE_TO_GBK[41816] := 16#9CDF;
   // UNICODE_TO_GBK[41817] := 16#F7AE;
   // UNICODE_TO_GBK[41818] := 16#9CE0;
   // UNICODE_TO_GBK[41819] := 16#F79F;
   // UNICODE_TO_GBK[41820] := 16#9CE1;
   // UNICODE_TO_GBK[41821] := 16#F7A0;
   // UNICODE_TO_GBK[41822] := 16#9CE2;
   // UNICODE_TO_GBK[41823] := 16#F7AF;
   // UNICODE_TO_GBK[41824] := 16#9CE3;
   // UNICODE_TO_GBK[41825] := 16#F840;
   // UNICODE_TO_GBK[41826] := 16#9CE4;
   // UNICODE_TO_GBK[41827] := 16#F841;
   // UNICODE_TO_GBK[41828] := 16#9CE5;
   // UNICODE_TO_GBK[41829] := 16#F842;
   // UNICODE_TO_GBK[41830] := 16#9CE6;
   // UNICODE_TO_GBK[41831] := 16#F843;
   // UNICODE_TO_GBK[41832] := 16#9CE7;
   // UNICODE_TO_GBK[41833] := 16#F844;
   // UNICODE_TO_GBK[41834] := 16#9CE8;
   // UNICODE_TO_GBK[41835] := 16#F845;
   // UNICODE_TO_GBK[41836] := 16#9CE9;
   // UNICODE_TO_GBK[41837] := 16#F846;
   // UNICODE_TO_GBK[41838] := 16#9CEA;
   // UNICODE_TO_GBK[41839] := 16#F847;
   // UNICODE_TO_GBK[41840] := 16#9CEB;
   // UNICODE_TO_GBK[41841] := 16#F848;
   // UNICODE_TO_GBK[41842] := 16#9CEC;
   // UNICODE_TO_GBK[41843] := 16#F849;
   // UNICODE_TO_GBK[41844] := 16#9CED;
   // UNICODE_TO_GBK[41845] := 16#F84A;
   // UNICODE_TO_GBK[41846] := 16#9CEE;
   // UNICODE_TO_GBK[41847] := 16#F84B;
   // UNICODE_TO_GBK[41848] := 16#9CEF;
   // UNICODE_TO_GBK[41849] := 16#F84C;
   // UNICODE_TO_GBK[41850] := 16#9CF0;
   // UNICODE_TO_GBK[41851] := 16#F84D;
   // UNICODE_TO_GBK[41852] := 16#9CF1;
   // UNICODE_TO_GBK[41853] := 16#F84E;
   // UNICODE_TO_GBK[41854] := 16#9CF2;
   // UNICODE_TO_GBK[41855] := 16#F84F;
   // UNICODE_TO_GBK[41856] := 16#9CF3;
   // UNICODE_TO_GBK[41857] := 16#F850;
   // UNICODE_TO_GBK[41858] := 16#9CF4;
   // UNICODE_TO_GBK[41859] := 16#F851;
   // UNICODE_TO_GBK[41860] := 16#9CF5;
   // UNICODE_TO_GBK[41861] := 16#F852;
   // UNICODE_TO_GBK[41862] := 16#9CF6;
   // UNICODE_TO_GBK[41863] := 16#F853;
   // UNICODE_TO_GBK[41864] := 16#9CF7;
   // UNICODE_TO_GBK[41865] := 16#F854;
   // UNICODE_TO_GBK[41866] := 16#9CF8;
   // UNICODE_TO_GBK[41867] := 16#F855;
   // UNICODE_TO_GBK[41868] := 16#9CF9;
   // UNICODE_TO_GBK[41869] := 16#F856;
   // UNICODE_TO_GBK[41870] := 16#9CFA;
   // UNICODE_TO_GBK[41871] := 16#F857;
   // UNICODE_TO_GBK[41872] := 16#9CFB;
   // UNICODE_TO_GBK[41873] := 16#F858;
   // UNICODE_TO_GBK[41874] := 16#9CFC;
   // UNICODE_TO_GBK[41875] := 16#F859;
   // UNICODE_TO_GBK[41876] := 16#9CFD;
   // UNICODE_TO_GBK[41877] := 16#F85A;
   // UNICODE_TO_GBK[41878] := 16#9CFE;
   // UNICODE_TO_GBK[41879] := 16#F85B;
   // UNICODE_TO_GBK[41880] := 16#9CFF;
   // UNICODE_TO_GBK[41881] := 16#F85C;
   // UNICODE_TO_GBK[41882] := 16#9D00;
   // UNICODE_TO_GBK[41883] := 16#F85D;
   // UNICODE_TO_GBK[41884] := 16#9D01;
   // UNICODE_TO_GBK[41885] := 16#F85E;
   // UNICODE_TO_GBK[41886] := 16#9D02;
   // UNICODE_TO_GBK[41887] := 16#F85F;
   // UNICODE_TO_GBK[41888] := 16#9D03;
   // UNICODE_TO_GBK[41889] := 16#F860;
   // UNICODE_TO_GBK[41890] := 16#9D04;
   // UNICODE_TO_GBK[41891] := 16#F861;
   // UNICODE_TO_GBK[41892] := 16#9D05;
   // UNICODE_TO_GBK[41893] := 16#F862;
   // UNICODE_TO_GBK[41894] := 16#9D06;
   // UNICODE_TO_GBK[41895] := 16#F863;
   // UNICODE_TO_GBK[41896] := 16#9D07;
   // UNICODE_TO_GBK[41897] := 16#F864;
   // UNICODE_TO_GBK[41898] := 16#9D08;
   // UNICODE_TO_GBK[41899] := 16#F865;
   // UNICODE_TO_GBK[41900] := 16#9D09;
   // UNICODE_TO_GBK[41901] := 16#F866;
   // UNICODE_TO_GBK[41902] := 16#9D0A;
   // UNICODE_TO_GBK[41903] := 16#F867;
   // UNICODE_TO_GBK[41904] := 16#9D0B;
   // UNICODE_TO_GBK[41905] := 16#F868;
   // UNICODE_TO_GBK[41906] := 16#9D0C;
   // UNICODE_TO_GBK[41907] := 16#F869;
   // UNICODE_TO_GBK[41908] := 16#9D0D;
   // UNICODE_TO_GBK[41909] := 16#F86A;
   // UNICODE_TO_GBK[41910] := 16#9D0E;
   // UNICODE_TO_GBK[41911] := 16#F86B;
   // UNICODE_TO_GBK[41912] := 16#9D0F;
   // UNICODE_TO_GBK[41913] := 16#F86C;
   // UNICODE_TO_GBK[41914] := 16#9D10;
   // UNICODE_TO_GBK[41915] := 16#F86D;
   // UNICODE_TO_GBK[41916] := 16#9D11;
   // UNICODE_TO_GBK[41917] := 16#F86E;
   // UNICODE_TO_GBK[41918] := 16#9D12;
   // UNICODE_TO_GBK[41919] := 16#F86F;
   // UNICODE_TO_GBK[41920] := 16#9D13;
   // UNICODE_TO_GBK[41921] := 16#F870;
   // UNICODE_TO_GBK[41922] := 16#9D14;
   // UNICODE_TO_GBK[41923] := 16#F871;
   // UNICODE_TO_GBK[41924] := 16#9D15;
   // UNICODE_TO_GBK[41925] := 16#F872;
   // UNICODE_TO_GBK[41926] := 16#9D16;
   // UNICODE_TO_GBK[41927] := 16#F873;
   // UNICODE_TO_GBK[41928] := 16#9D17;
   // UNICODE_TO_GBK[41929] := 16#F874;
   // UNICODE_TO_GBK[41930] := 16#9D18;
   // UNICODE_TO_GBK[41931] := 16#F875;
   // UNICODE_TO_GBK[41932] := 16#9D19;
   // UNICODE_TO_GBK[41933] := 16#F876;
   // UNICODE_TO_GBK[41934] := 16#9D1A;
   // UNICODE_TO_GBK[41935] := 16#F877;
   // UNICODE_TO_GBK[41936] := 16#9D1B;
   // UNICODE_TO_GBK[41937] := 16#F878;
   // UNICODE_TO_GBK[41938] := 16#9D1C;
   // UNICODE_TO_GBK[41939] := 16#F879;
   // UNICODE_TO_GBK[41940] := 16#9D1D;
   // UNICODE_TO_GBK[41941] := 16#F87A;
   // UNICODE_TO_GBK[41942] := 16#9D1E;
   // UNICODE_TO_GBK[41943] := 16#F87B;
   // UNICODE_TO_GBK[41944] := 16#9D1F;
   // UNICODE_TO_GBK[41945] := 16#F87C;
   // UNICODE_TO_GBK[41946] := 16#9D20;
   // UNICODE_TO_GBK[41947] := 16#F87D;
   // UNICODE_TO_GBK[41948] := 16#9D21;
   // UNICODE_TO_GBK[41949] := 16#F87E;
   // UNICODE_TO_GBK[41950] := 16#9D22;
   // UNICODE_TO_GBK[41951] := 16#F880;
   // UNICODE_TO_GBK[41952] := 16#9D23;
   // UNICODE_TO_GBK[41953] := 16#F881;
   // UNICODE_TO_GBK[41954] := 16#9D24;
   // UNICODE_TO_GBK[41955] := 16#F882;
   // UNICODE_TO_GBK[41956] := 16#9D25;
   // UNICODE_TO_GBK[41957] := 16#F883;
   // UNICODE_TO_GBK[41958] := 16#9D26;
   // UNICODE_TO_GBK[41959] := 16#F884;
   // UNICODE_TO_GBK[41960] := 16#9D27;
   // UNICODE_TO_GBK[41961] := 16#F885;
   // UNICODE_TO_GBK[41962] := 16#9D28;
   // UNICODE_TO_GBK[41963] := 16#F886;
   // UNICODE_TO_GBK[41964] := 16#9D29;
   // UNICODE_TO_GBK[41965] := 16#F887;
   // UNICODE_TO_GBK[41966] := 16#9D2A;
   // UNICODE_TO_GBK[41967] := 16#F888;
   // UNICODE_TO_GBK[41968] := 16#9D2B;
   // UNICODE_TO_GBK[41969] := 16#F889;
   // UNICODE_TO_GBK[41970] := 16#9D2C;
   // UNICODE_TO_GBK[41971] := 16#F88A;
   // UNICODE_TO_GBK[41972] := 16#9D2D;
   // UNICODE_TO_GBK[41973] := 16#F88B;
   // UNICODE_TO_GBK[41974] := 16#9D2E;
   // UNICODE_TO_GBK[41975] := 16#F88C;
   // UNICODE_TO_GBK[41976] := 16#9D2F;
   // UNICODE_TO_GBK[41977] := 16#F88D;
   // UNICODE_TO_GBK[41978] := 16#9D30;
   // UNICODE_TO_GBK[41979] := 16#F88E;
   // UNICODE_TO_GBK[41980] := 16#9D31;
   // UNICODE_TO_GBK[41981] := 16#F88F;
   // UNICODE_TO_GBK[41982] := 16#9D32;
   // UNICODE_TO_GBK[41983] := 16#F890;
   // UNICODE_TO_GBK[41984] := 16#9D33;
   // UNICODE_TO_GBK[41985] := 16#F891;
   // UNICODE_TO_GBK[41986] := 16#9D34;
   // UNICODE_TO_GBK[41987] := 16#F892;
   // UNICODE_TO_GBK[41988] := 16#9D35;
   // UNICODE_TO_GBK[41989] := 16#F893;
   // UNICODE_TO_GBK[41990] := 16#9D36;
   // UNICODE_TO_GBK[41991] := 16#F894;
   // UNICODE_TO_GBK[41992] := 16#9D37;
   // UNICODE_TO_GBK[41993] := 16#F895;
   // UNICODE_TO_GBK[41994] := 16#9D38;
   // UNICODE_TO_GBK[41995] := 16#F896;
   // UNICODE_TO_GBK[41996] := 16#9D39;
   // UNICODE_TO_GBK[41997] := 16#F897;
   // UNICODE_TO_GBK[41998] := 16#9D3A;
   // UNICODE_TO_GBK[41999] := 16#F898;
   // UNICODE_TO_GBK[42000] := 16#9D3B;
   // UNICODE_TO_GBK[42001] := 16#F899;
   // UNICODE_TO_GBK[42002] := 16#9D3C;
   // UNICODE_TO_GBK[42003] := 16#F89A;
   // UNICODE_TO_GBK[42004] := 16#9D3D;
   // UNICODE_TO_GBK[42005] := 16#F89B;
   // UNICODE_TO_GBK[42006] := 16#9D3E;
   // UNICODE_TO_GBK[42007] := 16#F89C;
   // UNICODE_TO_GBK[42008] := 16#9D3F;
   // UNICODE_TO_GBK[42009] := 16#F89D;
   // UNICODE_TO_GBK[42010] := 16#9D40;
   // UNICODE_TO_GBK[42011] := 16#F89E;
   // UNICODE_TO_GBK[42012] := 16#9D41;
   // UNICODE_TO_GBK[42013] := 16#F89F;
   // UNICODE_TO_GBK[42014] := 16#9D42;
   // UNICODE_TO_GBK[42015] := 16#F8A0;
   // UNICODE_TO_GBK[42016] := 16#9D43;
   // UNICODE_TO_GBK[42017] := 16#F940;
   // UNICODE_TO_GBK[42018] := 16#9D44;
   // UNICODE_TO_GBK[42019] := 16#F941;
   // UNICODE_TO_GBK[42020] := 16#9D45;
   // UNICODE_TO_GBK[42021] := 16#F942;
   // UNICODE_TO_GBK[42022] := 16#9D46;
   // UNICODE_TO_GBK[42023] := 16#F943;
   // UNICODE_TO_GBK[42024] := 16#9D47;
   // UNICODE_TO_GBK[42025] := 16#F944;
   // UNICODE_TO_GBK[42026] := 16#9D48;
   // UNICODE_TO_GBK[42027] := 16#F945;
   // UNICODE_TO_GBK[42028] := 16#9D49;
   // UNICODE_TO_GBK[42029] := 16#F946;
   // UNICODE_TO_GBK[42030] := 16#9D4A;
   // UNICODE_TO_GBK[42031] := 16#F947;
   // UNICODE_TO_GBK[42032] := 16#9D4B;
   // UNICODE_TO_GBK[42033] := 16#F948;
   // UNICODE_TO_GBK[42034] := 16#9D4C;
   // UNICODE_TO_GBK[42035] := 16#F949;
   // UNICODE_TO_GBK[42036] := 16#9D4D;
   // UNICODE_TO_GBK[42037] := 16#F94A;
   // UNICODE_TO_GBK[42038] := 16#9D4E;
   // UNICODE_TO_GBK[42039] := 16#F94B;
   // UNICODE_TO_GBK[42040] := 16#9D4F;
   // UNICODE_TO_GBK[42041] := 16#F94C;
   // UNICODE_TO_GBK[42042] := 16#9D50;
   // UNICODE_TO_GBK[42043] := 16#F94D;
   // UNICODE_TO_GBK[42044] := 16#9D51;
   // UNICODE_TO_GBK[42045] := 16#F94E;
   // UNICODE_TO_GBK[42046] := 16#9D52;
   // UNICODE_TO_GBK[42047] := 16#F94F;
   // UNICODE_TO_GBK[42048] := 16#9D53;
   // UNICODE_TO_GBK[42049] := 16#F950;
   // UNICODE_TO_GBK[42050] := 16#9D54;
   // UNICODE_TO_GBK[42051] := 16#F951;
   // UNICODE_TO_GBK[42052] := 16#9D55;
   // UNICODE_TO_GBK[42053] := 16#F952;
   // UNICODE_TO_GBK[42054] := 16#9D56;
   // UNICODE_TO_GBK[42055] := 16#F953;
   // UNICODE_TO_GBK[42056] := 16#9D57;
   // UNICODE_TO_GBK[42057] := 16#F954;
   // UNICODE_TO_GBK[42058] := 16#9D58;
   // UNICODE_TO_GBK[42059] := 16#F955;
   // UNICODE_TO_GBK[42060] := 16#9D59;
   // UNICODE_TO_GBK[42061] := 16#F956;
   // UNICODE_TO_GBK[42062] := 16#9D5A;
   // UNICODE_TO_GBK[42063] := 16#F957;
   // UNICODE_TO_GBK[42064] := 16#9D5B;
   // UNICODE_TO_GBK[42065] := 16#F958;
   // UNICODE_TO_GBK[42066] := 16#9D5C;
   // UNICODE_TO_GBK[42067] := 16#F959;
   // UNICODE_TO_GBK[42068] := 16#9D5D;
   // UNICODE_TO_GBK[42069] := 16#F95A;
   // UNICODE_TO_GBK[42070] := 16#9D5E;
   // UNICODE_TO_GBK[42071] := 16#F95B;
   // UNICODE_TO_GBK[42072] := 16#9D5F;
   // UNICODE_TO_GBK[42073] := 16#F95C;
   // UNICODE_TO_GBK[42074] := 16#9D60;
   // UNICODE_TO_GBK[42075] := 16#F95D;
   // UNICODE_TO_GBK[42076] := 16#9D61;
   // UNICODE_TO_GBK[42077] := 16#F95E;
   // UNICODE_TO_GBK[42078] := 16#9D62;
   // UNICODE_TO_GBK[42079] := 16#F95F;
   // UNICODE_TO_GBK[42080] := 16#9D63;
   // UNICODE_TO_GBK[42081] := 16#F960;
   // UNICODE_TO_GBK[42082] := 16#9D64;
   // UNICODE_TO_GBK[42083] := 16#F961;
   // UNICODE_TO_GBK[42084] := 16#9D65;
   // UNICODE_TO_GBK[42085] := 16#F962;
   // UNICODE_TO_GBK[42086] := 16#9D66;
   // UNICODE_TO_GBK[42087] := 16#F963;
   // UNICODE_TO_GBK[42088] := 16#9D67;
   // UNICODE_TO_GBK[42089] := 16#F964;
   // UNICODE_TO_GBK[42090] := 16#9D68;
   // UNICODE_TO_GBK[42091] := 16#F965;
   // UNICODE_TO_GBK[42092] := 16#9D69;
   // UNICODE_TO_GBK[42093] := 16#F966;
   // UNICODE_TO_GBK[42094] := 16#9D6A;
   // UNICODE_TO_GBK[42095] := 16#F967;
   // UNICODE_TO_GBK[42096] := 16#9D6B;
   // UNICODE_TO_GBK[42097] := 16#F968;
   // UNICODE_TO_GBK[42098] := 16#9D6C;
   // UNICODE_TO_GBK[42099] := 16#F969;
   // UNICODE_TO_GBK[42100] := 16#9D6D;
   // UNICODE_TO_GBK[42101] := 16#F96A;
   // UNICODE_TO_GBK[42102] := 16#9D6E;
   // UNICODE_TO_GBK[42103] := 16#F96B;
   // UNICODE_TO_GBK[42104] := 16#9D6F;
   // UNICODE_TO_GBK[42105] := 16#F96C;
   // UNICODE_TO_GBK[42106] := 16#9D70;
   // UNICODE_TO_GBK[42107] := 16#F96D;
   // UNICODE_TO_GBK[42108] := 16#9D71;
   // UNICODE_TO_GBK[42109] := 16#F96E;
   // UNICODE_TO_GBK[42110] := 16#9D72;
   // UNICODE_TO_GBK[42111] := 16#F96F;
   // UNICODE_TO_GBK[42112] := 16#9D73;
   // UNICODE_TO_GBK[42113] := 16#F970;
   // UNICODE_TO_GBK[42114] := 16#9D74;
   // UNICODE_TO_GBK[42115] := 16#F971;
   // UNICODE_TO_GBK[42116] := 16#9D75;
   // UNICODE_TO_GBK[42117] := 16#F972;
   // UNICODE_TO_GBK[42118] := 16#9D76;
   // UNICODE_TO_GBK[42119] := 16#F973;
   // UNICODE_TO_GBK[42120] := 16#9D77;
   // UNICODE_TO_GBK[42121] := 16#F974;
   // UNICODE_TO_GBK[42122] := 16#9D78;
   // UNICODE_TO_GBK[42123] := 16#F975;
   // UNICODE_TO_GBK[42124] := 16#9D79;
   // UNICODE_TO_GBK[42125] := 16#F976;
   // UNICODE_TO_GBK[42126] := 16#9D7A;
   // UNICODE_TO_GBK[42127] := 16#F977;
   // UNICODE_TO_GBK[42128] := 16#9D7B;
   // UNICODE_TO_GBK[42129] := 16#F978;
   // UNICODE_TO_GBK[42130] := 16#9D7C;
   // UNICODE_TO_GBK[42131] := 16#F979;
   // UNICODE_TO_GBK[42132] := 16#9D7D;
   // UNICODE_TO_GBK[42133] := 16#F97A;
   // UNICODE_TO_GBK[42134] := 16#9D7E;
   // UNICODE_TO_GBK[42135] := 16#F97B;
   // UNICODE_TO_GBK[42136] := 16#9D7F;
   // UNICODE_TO_GBK[42137] := 16#F97C;
   // UNICODE_TO_GBK[42138] := 16#9D80;
   // UNICODE_TO_GBK[42139] := 16#F97D;
   // UNICODE_TO_GBK[42140] := 16#9D81;
   // UNICODE_TO_GBK[42141] := 16#F97E;
   // UNICODE_TO_GBK[42142] := 16#9D82;
   // UNICODE_TO_GBK[42143] := 16#F980;
   // UNICODE_TO_GBK[42144] := 16#9D83;
   // UNICODE_TO_GBK[42145] := 16#F981;
   // UNICODE_TO_GBK[42146] := 16#9D84;
   // UNICODE_TO_GBK[42147] := 16#F982;
   // UNICODE_TO_GBK[42148] := 16#9D85;
   // UNICODE_TO_GBK[42149] := 16#F983;
   // UNICODE_TO_GBK[42150] := 16#9D86;
   // UNICODE_TO_GBK[42151] := 16#F984;
   // UNICODE_TO_GBK[42152] := 16#9D87;
   // UNICODE_TO_GBK[42153] := 16#F985;
   // UNICODE_TO_GBK[42154] := 16#9D88;
   // UNICODE_TO_GBK[42155] := 16#F986;
   // UNICODE_TO_GBK[42156] := 16#9D89;
   // UNICODE_TO_GBK[42157] := 16#F987;
   // UNICODE_TO_GBK[42158] := 16#9D8A;
   // UNICODE_TO_GBK[42159] := 16#F988;
   // UNICODE_TO_GBK[42160] := 16#9D8B;
   // UNICODE_TO_GBK[42161] := 16#F989;
   // UNICODE_TO_GBK[42162] := 16#9D8C;
   // UNICODE_TO_GBK[42163] := 16#F98A;
   // UNICODE_TO_GBK[42164] := 16#9D8D;
   // UNICODE_TO_GBK[42165] := 16#F98B;
   // UNICODE_TO_GBK[42166] := 16#9D8E;
   // UNICODE_TO_GBK[42167] := 16#F98C;
   // UNICODE_TO_GBK[42168] := 16#9D8F;
   // UNICODE_TO_GBK[42169] := 16#F98D;
   // UNICODE_TO_GBK[42170] := 16#9D90;
   // UNICODE_TO_GBK[42171] := 16#F98E;
   // UNICODE_TO_GBK[42172] := 16#9D91;
   // UNICODE_TO_GBK[42173] := 16#F98F;
   // UNICODE_TO_GBK[42174] := 16#9D92;
   // UNICODE_TO_GBK[42175] := 16#F990;
   // UNICODE_TO_GBK[42176] := 16#9D93;
   // UNICODE_TO_GBK[42177] := 16#F991;
   // UNICODE_TO_GBK[42178] := 16#9D94;
   // UNICODE_TO_GBK[42179] := 16#F992;
   // UNICODE_TO_GBK[42180] := 16#9D95;
   // UNICODE_TO_GBK[42181] := 16#F993;
   // UNICODE_TO_GBK[42182] := 16#9D96;
   // UNICODE_TO_GBK[42183] := 16#F994;
   // UNICODE_TO_GBK[42184] := 16#9D97;
   // UNICODE_TO_GBK[42185] := 16#F995;
   // UNICODE_TO_GBK[42186] := 16#9D98;
   // UNICODE_TO_GBK[42187] := 16#F996;
   // UNICODE_TO_GBK[42188] := 16#9D99;
   // UNICODE_TO_GBK[42189] := 16#F997;
   // UNICODE_TO_GBK[42190] := 16#9D9A;
   // UNICODE_TO_GBK[42191] := 16#F998;
   // UNICODE_TO_GBK[42192] := 16#9D9B;
   // UNICODE_TO_GBK[42193] := 16#F999;
   // UNICODE_TO_GBK[42194] := 16#9D9C;
   // UNICODE_TO_GBK[42195] := 16#F99A;
   // UNICODE_TO_GBK[42196] := 16#9D9D;
   // UNICODE_TO_GBK[42197] := 16#F99B;
   // UNICODE_TO_GBK[42198] := 16#9D9E;
   // UNICODE_TO_GBK[42199] := 16#F99C;
   // UNICODE_TO_GBK[42200] := 16#9D9F;
   // UNICODE_TO_GBK[42201] := 16#F99D;
   // UNICODE_TO_GBK[42202] := 16#9DA0;
   // UNICODE_TO_GBK[42203] := 16#F99E;
   // UNICODE_TO_GBK[42204] := 16#9DA1;
   // UNICODE_TO_GBK[42205] := 16#F99F;
   // UNICODE_TO_GBK[42206] := 16#9DA2;
   // UNICODE_TO_GBK[42207] := 16#F9A0;
   // UNICODE_TO_GBK[42208] := 16#9DA3;
   // UNICODE_TO_GBK[42209] := 16#FA40;
   // UNICODE_TO_GBK[42210] := 16#9DA4;
   // UNICODE_TO_GBK[42211] := 16#FA41;
   // UNICODE_TO_GBK[42212] := 16#9DA5;
   // UNICODE_TO_GBK[42213] := 16#FA42;
   // UNICODE_TO_GBK[42214] := 16#9DA6;
   // UNICODE_TO_GBK[42215] := 16#FA43;
   // UNICODE_TO_GBK[42216] := 16#9DA7;
   // UNICODE_TO_GBK[42217] := 16#FA44;
   // UNICODE_TO_GBK[42218] := 16#9DA8;
   // UNICODE_TO_GBK[42219] := 16#FA45;
   // UNICODE_TO_GBK[42220] := 16#9DA9;
   // UNICODE_TO_GBK[42221] := 16#FA46;
   // UNICODE_TO_GBK[42222] := 16#9DAA;
   // UNICODE_TO_GBK[42223] := 16#FA47;
   // UNICODE_TO_GBK[42224] := 16#9DAB;
   // UNICODE_TO_GBK[42225] := 16#FA48;
   // UNICODE_TO_GBK[42226] := 16#9DAC;
   // UNICODE_TO_GBK[42227] := 16#FA49;
   // UNICODE_TO_GBK[42228] := 16#9DAD;
   // UNICODE_TO_GBK[42229] := 16#FA4A;
   // UNICODE_TO_GBK[42230] := 16#9DAE;
   // UNICODE_TO_GBK[42231] := 16#FA4B;
   // UNICODE_TO_GBK[42232] := 16#9DAF;
   // UNICODE_TO_GBK[42233] := 16#FA4C;
   // UNICODE_TO_GBK[42234] := 16#9DB0;
   // UNICODE_TO_GBK[42235] := 16#FA4D;
   // UNICODE_TO_GBK[42236] := 16#9DB1;
   // UNICODE_TO_GBK[42237] := 16#FA4E;
   // UNICODE_TO_GBK[42238] := 16#9DB2;
   // UNICODE_TO_GBK[42239] := 16#FA4F;
   // UNICODE_TO_GBK[42240] := 16#9DB3;
   // UNICODE_TO_GBK[42241] := 16#FA50;
   // UNICODE_TO_GBK[42242] := 16#9DB4;
   // UNICODE_TO_GBK[42243] := 16#FA51;
   // UNICODE_TO_GBK[42244] := 16#9DB5;
   // UNICODE_TO_GBK[42245] := 16#FA52;
   // UNICODE_TO_GBK[42246] := 16#9DB6;
   // UNICODE_TO_GBK[42247] := 16#FA53;
   // UNICODE_TO_GBK[42248] := 16#9DB7;
   // UNICODE_TO_GBK[42249] := 16#FA54;
   // UNICODE_TO_GBK[42250] := 16#9DB8;
   // UNICODE_TO_GBK[42251] := 16#FA55;
   // UNICODE_TO_GBK[42252] := 16#9DB9;
   // UNICODE_TO_GBK[42253] := 16#FA56;
   // UNICODE_TO_GBK[42254] := 16#9DBA;
   // UNICODE_TO_GBK[42255] := 16#FA57;
   // UNICODE_TO_GBK[42256] := 16#9DBB;
   // UNICODE_TO_GBK[42257] := 16#FA58;
   // UNICODE_TO_GBK[42258] := 16#9DBC;
   // UNICODE_TO_GBK[42259] := 16#FA59;
   // UNICODE_TO_GBK[42260] := 16#9DBD;
   // UNICODE_TO_GBK[42261] := 16#FA5A;
   // UNICODE_TO_GBK[42262] := 16#9DBE;
   // UNICODE_TO_GBK[42263] := 16#FA5B;
   // UNICODE_TO_GBK[42264] := 16#9DBF;
   // UNICODE_TO_GBK[42265] := 16#FA5C;
   // UNICODE_TO_GBK[42266] := 16#9DC0;
   // UNICODE_TO_GBK[42267] := 16#FA5D;
   // UNICODE_TO_GBK[42268] := 16#9DC1;
   // UNICODE_TO_GBK[42269] := 16#FA5E;
   // UNICODE_TO_GBK[42270] := 16#9DC2;
   // UNICODE_TO_GBK[42271] := 16#FA5F;
   // UNICODE_TO_GBK[42272] := 16#9DC3;
   // UNICODE_TO_GBK[42273] := 16#FA60;
   // UNICODE_TO_GBK[42274] := 16#9DC4;
   // UNICODE_TO_GBK[42275] := 16#FA61;
   // UNICODE_TO_GBK[42276] := 16#9DC5;
   // UNICODE_TO_GBK[42277] := 16#FA62;
   // UNICODE_TO_GBK[42278] := 16#9DC6;
   // UNICODE_TO_GBK[42279] := 16#FA63;
   // UNICODE_TO_GBK[42280] := 16#9DC7;
   // UNICODE_TO_GBK[42281] := 16#FA64;
   // UNICODE_TO_GBK[42282] := 16#9DC8;
   // UNICODE_TO_GBK[42283] := 16#FA65;
   // UNICODE_TO_GBK[42284] := 16#9DC9;
   // UNICODE_TO_GBK[42285] := 16#FA66;
   // UNICODE_TO_GBK[42286] := 16#9DCA;
   // UNICODE_TO_GBK[42287] := 16#FA67;
   // UNICODE_TO_GBK[42288] := 16#9DCB;
   // UNICODE_TO_GBK[42289] := 16#FA68;
   // UNICODE_TO_GBK[42290] := 16#9DCC;
   // UNICODE_TO_GBK[42291] := 16#FA69;
   // UNICODE_TO_GBK[42292] := 16#9DCD;
   // UNICODE_TO_GBK[42293] := 16#FA6A;
   // UNICODE_TO_GBK[42294] := 16#9DCE;
   // UNICODE_TO_GBK[42295] := 16#FA6B;
   // UNICODE_TO_GBK[42296] := 16#9DCF;
   // UNICODE_TO_GBK[42297] := 16#FA6C;
   // UNICODE_TO_GBK[42298] := 16#9DD0;
   // UNICODE_TO_GBK[42299] := 16#FA6D;
   // UNICODE_TO_GBK[42300] := 16#9DD1;
   // UNICODE_TO_GBK[42301] := 16#FA6E;
   // UNICODE_TO_GBK[42302] := 16#9DD2;
   // UNICODE_TO_GBK[42303] := 16#FA6F;
   // UNICODE_TO_GBK[42304] := 16#9DD3;
   // UNICODE_TO_GBK[42305] := 16#FA70;
   // UNICODE_TO_GBK[42306] := 16#9DD4;
   // UNICODE_TO_GBK[42307] := 16#FA71;
   // UNICODE_TO_GBK[42308] := 16#9DD5;
   // UNICODE_TO_GBK[42309] := 16#FA72;
   // UNICODE_TO_GBK[42310] := 16#9DD6;
   // UNICODE_TO_GBK[42311] := 16#FA73;
   // UNICODE_TO_GBK[42312] := 16#9DD7;
   // UNICODE_TO_GBK[42313] := 16#FA74;
   // UNICODE_TO_GBK[42314] := 16#9DD8;
   // UNICODE_TO_GBK[42315] := 16#FA75;
   // UNICODE_TO_GBK[42316] := 16#9DD9;
   // UNICODE_TO_GBK[42317] := 16#FA76;
   // UNICODE_TO_GBK[42318] := 16#9DDA;
   // UNICODE_TO_GBK[42319] := 16#FA77;
   // UNICODE_TO_GBK[42320] := 16#9DDB;
   // UNICODE_TO_GBK[42321] := 16#FA78;
   // UNICODE_TO_GBK[42322] := 16#9DDC;
   // UNICODE_TO_GBK[42323] := 16#FA79;
   // UNICODE_TO_GBK[42324] := 16#9DDD;
   // UNICODE_TO_GBK[42325] := 16#FA7A;
